CR130_LH_Rot_Cyl(
	Auto:=OP130_AutoSelected , 
	Manual:=OP130_ManualSelected, 
	ErrorActive:=OP130_ErrorActive , 
	ResetPB:= , 
	Sensor1:= I130_LH_ROTRY_180_DEGI1300_1, 
	Sensor2:= I130_LH_ROTRY_0_DEGI1300_0, 
	ManualPB1:= , 
	ManualPB2:= , 
	AutoCmd1:= , 
	AutoCmd2:= , 
	OperationEnable:=OperationEnable , 
	SafeHome:= , 
	SafeWork:= , 
	HomingCmd1:= , 
	Pulse_1Sec:=Pulse_Block.Q1Hz , 
	BlinkingBit:= , 
	TimeOut1:=10 , 
	TimeOut2:=10 , 
	TimeOut3:=10 , 
	Solenoid1=> O130_LH_ROTRY_180_DEG_Q1340_1, 
	Solenoid2=> O130_LH_ROTRY_0_DEG_Q1340_0, 
	AlarmSensor1=>berror[1201] , 
	AlarmSensor2=>berror[1202] , 
	AlarmSolenoid1=>berror[1205] , 
	AlarmSolenoid2=>berror[1206] , 
	AllSignal=>berror[1207] , 
	AlarmPresent=> , 
	Position1=> , 
	Position2=> , 
	HomeSensorBlink=> , 
	WorkSensorBlink=> , 
	Status:=CR130_LH_Rotart_Cyl_Stats );
	
//RH Rotary Cylinder


//move ZERO to STATUS
OP130_GVL.CR130_RH_Rotart_Cyl_Status:=0;



//Reset Auto Cmd IN Manual Mode & Homing
IF ( OP130_HomeRunning) THEN
	CR130_RH_Rot_Cyl.AutoCmd1:=FALSE;
	CR130_RH_Rot_Cyl.AutoCmd2:=FALSE;		
END_IF

// Safe Home
IF SR130_stManualModeAxis_RH_Vert_Servo.actualPosition >=57.0 THEN 
	CR130_RH_Rot_Cyl.SafeHome:= TRUE ;
	ELSE 
		CR130_RH_Rot_Cyl.SafeHome:= FALSE ;
	END_IF
// Safe Work
IF SR130_stManualModeAxis_RH_Vert_Servo.actualPosition >=57.0   THEN 
	CR130_RH_Rot_Cyl.Safework:= TRUE ;
	ELSE 
		CR130_RH_Rot_Cyl.Safework:= FALSE ;
	END_IF
	
// Manual PB  Cyl Mapping
IF (OP130_HMI_RH_Rotary_Cyl_Home_PB=TRUE) THEN
	CR130_RH_Rot_Cyl.ManualPB1:=TRUE;
	ELSE 
		CR130_RH_Rot_Cyl.ManualPB1:=FALSE;
	END_IF
	
IF (OP130_HMI_RH_Rotary_Cyl_Work_PB=TRUE) THEN
	CR130_RH_Rot_Cyl.ManualPB2:=TRUE;
	ELSE 
		CR130_RH_Rot_Cyl.ManualPB2:=FALSE;
	END_IF


	
CR130_RH_Rot_Cyl(
	Auto:=OP130_AutoSelected , 
	Manual:=OP130_ManualSelected , 
	ErrorActive:=OP130_ErrorActive , 
	ResetPB:= , 
	Sensor1:= I130_RH_ROTRY_180_DEGI1300_3, 
	Sensor2:= I130_RH_ROTRY_0_DEGI1300_2, 
	ManualPB1:= , 
	ManualPB2:= , 
	AutoCmd1:= , 
	AutoCmd2:= , 
	OperationEnable:=OperationEnable , 
	SafeHome:= , 
	SafeWork:= , 
	HomingCmd1:= , 
	Pulse_1Sec:=Pulse_Block.Q1Hz  , 
	BlinkingBit:= , 
	TimeOut1:=10 , 
	TimeOut2:=10 , 
	TimeOut3:=10 , 
	Solenoid1=> O130_RH_ROTRY_180_DEG_Q1340_3, 
	Solenoid2=> O130_RH_ROTRY_0_DEG_Q1340_2, 
	AlarmSensor1=>berror[1208] , 
	AlarmSensor2=>berror[1209] , 
	AlarmSolenoid1=>berror[1210] , 
	AlarmSolenoid2=>berror[1211] , 
	AllSignal=>berror[1212] , 
	AlarmPresent=> , 
	Position1=> , 
	Position2=> , 
	HomeSensorBlink=> , 
	WorkSensorBlink=> , 
	Status:=CR130_RH_Rotart_Cyl_Stats );
	
//LH Vertical Slide Servo

// Servo Safe To move
IF (SR130_stManualModeAxis_LH_Vert_Servo.actualPosition < 57.0 AND CR130_LH_Rot_Cyl.Position2)  THEN 
	OP130_LH_Servo_Safety:= FALSE;
	ELSE
	OP130_LH_Servo_Safety:= TRUE;	
	END_IF



//SR130_LH_Vert_Servo(
//	bAxis1_Ref_Switch:= , 
//	bInit:= , 
//	bErrorReset:= , 
//	bEnable:= , 
//	bMoveVelocity:= , 
//	bHalt:= , 
//	bManualMode:= , 
//	fHomePos:=SR130_LH_Servo_Control.Reference_Position , 
//	fOverride:= , 
//	fTargetPosition:= , 
//	fTargetVelocity:= , 
//	fAcc:= , 
//	fDec:= , 
//	Axis:=SR130_RH_Vert_Servo_Axis, 
//	bHome:=SR130_LH_Servo_Control.Reference_Start , 
//	bSetPosition:=SR130_LH_Servo_Control.BsetPos , 
//	bMoveAbsolute:=SR130_LH_Servo_Control.ABSmove_Start , 
//	bMoveRelative:=SR130_LH_Servo_Control.RELmove_Start , 
//	stManualModeAxis:=SR130_stManualModeAxis_LH_Vert_Servo, 
//	sAxisState=>SR130_LH_Servo_Control.Axis_State , 
//	bAxis_ready=>SR130_LH_Servo_Control.Axis_ready , 
//	bAxisInPosition=>SR130_LH_Servo_Control.Axis_In_Pos , 
//	bAxisError=>SR130_LH_Servo_Control.Axis_Error , 
//	bAxisEnabled=>SR130_LH_Servo_Control.Axis_Enabled , 
//	bAxisHomed=>SR130_LH_Servo_Control.Axis_reference , 
//	bSetPositionDone=> , 
//	bHaltDone=> , 
//	bSTOPDone=> , 
//	bHomeDone=> , 
//	bDone=> );

	
	//LH Vertical Servo 1
	SR130_LH_Vert_Servo(
	bAxis1_Ref_Switch:= , 
	bInit:= , 
	bErrorReset:=OP130_HMI_Reset OR Servo_Reset , 
	bEnable:= OperationEnable, 
	bMoveVelocity:= , 
	bHalt:= , 
	bManualMode:=OP130_ManualSelected , 
	fHomePos:= , 
	fOverride:= , 
	fTargetPosition:=SR130_LH_Servo_Control.Position , 
	fTargetVelocity:=SR130_LH_Servo_Control.Velocity, 
	fAcc:= , 
	fDec:= ,
	Servo_High_Limit:= SR130_LH_Vert_Servo_Max_Limit,	
	Servo_Low_Limit:=SR130_LH_Vert_Servo_Min_Lim,	 	
	WARNING_LIMIT:=1,
	TORQUE_LIMIT=>,	 
	Safe_move_Conditions:=OP130_LH_Servo_Safety , 
	Axis:= SR130_LH_Vert_Servo_Axis, 
	HME_WRITE_ADD:= 16#5013,	
	bHome:= SR130_LH_Servo_Control.Reference_Start, 
	bSetPosition:=SR130_LH_Servo_Control.BsetPos , 
	bMoveAbsolute:= SR130_LH_Servo_Control.ABSmove_Start , 
	bMoveRelative:=SR130_LH_Servo_Control.RELmove_Start , 
	bMoveTorque:=SR130_LH_Servo_Control.Torque_mode_Start , 
	stManualModeAxis:=SR130_stManualModeAxis_LH_Vert_Servo , 
	bmove_home:=SR130_LH_Servo_Control.Axis_Home_Cmd , 
	sAxisState=>SR130_LH_Servo_Control.Axis_State , 
	bAxis_ready=>SR130_LH_Servo_Control.Axis_ready , 
	bAxisInPosition=>SR130_LH_Servo_Control.Axis_In_Pos , 
	bAxisError=>berror[1250] , 
	bAxisEnabled=> SR130_LH_Servo_Control.Axis_Enabled, 
	bAxisHomed=>SR130_LH_Servo_Control.Axis_reference  , 
	bSetPositionDone=> , 
	bHaltDone=> SR130_LH_Servo_Control.Axis_Halted, 
	bSTOPDone=> SR130_LH_Servo_Control.Axis_Stopped, 
	bHomeDone=> , 
	bDone=> , 
	bTorqueReached=>SR130_LH_Servo_Control.Trq_reached , 
	bsafe_to_move=>SR130_LH_Servo_Control.Safe_To_Move , 
	baxis_in_home_pos=>SR130_LH_Servo_Control.Axis_In_Home , 
	bABS_Pos_done=> , 
	Actual_position=>SR130_LH_Servo_Control.Actual_Position, 
	Actual_velocity=>SR130_LH_Servo_Control.Actual_Velocity , 
	Actual_Torque=>SR130_LH_Servo_Control.Actual_Torque );
	

	
	//RH Vertical Slide Servo

// Servo Safe To move
IF (SR130_stManualModeAxis_RH_Vert_Servo.actualPosition < 57.0 AND CR130_RH_Rot_Cyl.Position2) THEN 
	OP130_RH_Servo_Safety:= FALSE;
	ELSE
	OP130_RH_Servo_Safety:= TRUE;	
	END_IF


//SR130_RH_Vert_Servo(
//	bAxis1_Ref_Switch:= , 
//	bInit:= , 
//	bErrorReset:= , 
//	bEnable:= , 
//	bMoveVelocity:= , 
//	bHalt:= , 
//	bManualMode:= , 
//	fHomePos:=SR130_RH_Servo_Control.Reference_Position , 
//	fOverride:= , 
//	fTargetPosition:= , 
//	fTargetVelocity:= , 
//	fAcc:= , 
//	fDec:= , 
//	Axis:=SR130_LH_Vert_Servo_Axis , 
//	bHome:=SR130_RH_Servo_Control.Reference_Start , 
//	bSetPosition:=SR130_RH_Servo_Control.BsetPos , 
//	bMoveAbsolute:=SR130_RH_Servo_Control.ABSmove_Start , 
//	bMoveRelative:=SR130_RH_Servo_Control.RELmove_Start , 
//	stManualModeAxis:=SR130_stManualModeAxis_RH_Vert_Servo , 
//	sAxisState=>SR130_RH_Servo_Control.Axis_State , 
//	bAxis_ready=>SR130_RH_Servo_Control.Axis_ready , 
//	bAxisInPosition=>SR130_RH_Servo_Control.Axis_In_Pos , 
//	bAxisError=>SR130_RH_Servo_Control.Axis_Error , 
//	bAxisEnabled=>SR130_RH_Servo_Control.Axis_Enabled , 
//	bAxisHomed=>SR130_RH_Servo_Control.Axis_reference , 
//	bSetPositionDone=> , 
//	bHaltDone=> , 
//	bSTOPDone=> , 
//	bHomeDone=> , 
//	bDone=> );
	
//RH Vert Servo 1

SR130_RH_Vert_Servo(
	bAxis1_Ref_Switch:= , 
	bInit:= , 
	bErrorReset:=OP130_HMI_Reset OR Servo_Reset , 
	bEnable:= OperationEnable , 
	bMoveVelocity:= , 
	bHalt:= , 
	bManualMode:=OP130_ManualSelected , 
	fHomePos:=SR130_RH_Servo_Control.Reference_Position , 
	fOverride:= , 
	fTargetPosition:= SR130_RH_Servo_Control.Position , 
	fTargetVelocity:=SR130_RH_Servo_Control.Velocity , 
	fAcc:= , 
	fDec:= ,
	Servo_High_Limit:= SR130_LH_Vert_Servo_Max_Limit,	
	Servo_Low_Limit:=SR130_LH_Vert_Servo_Min_Lim,	 	
	WARNING_LIMIT:=1,
	Actual_Torque=>SR130_RH_Servo_Control.Actual_Torque  ,
	Actual_position=> ,
    Actual_velocity=> ,
	TORQUE_LIMIT=>,	 
	Safe_move_Conditions:=OP130_RH_Servo_Safety , 
	Axis:= SR130_RH_Vert_Servo_Axis, 
	HME_WRITE_ADD:= 16#5012,	
	bHome:=SR130_LH_Servo_Control.Reference_Start , 
	bSetPosition:= SR130_RH_Servo_Control.BsetPos, 
	bMoveAbsolute:= SR130_RH_Servo_Control.ABSmove_Start, 
	bMoveRelative:=SR130_RH_Servo_Control.RELmove_Start , 
	bMoveTorque:=SR130_RH_Servo_Control.Torque_mode_Start , 
	stManualModeAxis:=SR130_stManualModeAxis_RH_Vert_Servo , 
	bmove_home:=SR130_RH_Servo_Control.Axis_Home_Cmd , 
	sAxisState=>SR130_RH_Servo_Control.Axis_State , 
	bAxis_ready=>SR130_RH_Servo_Control.Axis_ready  , 
	bAxisInPosition=>SR130_RH_Servo_Control.Axis_In_Pos , 
	bAxisError=>berror[1251] , 
	bAxisEnabled=>SR130_RH_Servo_Control.Axis_Enabled , 
	bAxisHomed=>SR130_RH_Servo_Control.Axis_reference , 
	bSetPositionDone=> , 
	bHaltDone=>SR130_RH_Servo_Control.Axis_Halted , 
	bSTOPDone=>SR130_RH_Servo_Control.Axis_Stopped , 
	bHomeDone=> , 
	bDone=> , 
	bTorqueReached=> SR130_RH_Servo_Control.Trq_reached, 
	bsafe_to_move=> SR130_RH_Servo_Control.Safe_To_Move, 
	baxis_in_home_pos=>SR130_RH_Servo_Control.Axis_In_Home , 
	bABS_Pos_done=> , 
	Actual_position=>SR130_RH_Servo_Control.Actual_Position , 
	Actual_velocity=>SR130_RH_Servo_Control.Actual_Velocity , 
	Actual_Torque=> SR130_RH_Servo_Control.Actual_Torque);
	
	// Clamping Stepper 
	// Servo Safe To move
IF (TRUE) THEN 
	SR130_RH_Servo_Control.Safe_To_Move:= TRUE;
END_IF
IF MANUAL_SELECTED THEN
	SR130_stManualModeAxis_Clamp_Stepper.targetVelocity:=50;
END_IF

SR130_Clm_Stepper(														// FESTO GUIDE GRIPPER
	bAxis1_Ref_Switch:= , 
	bInit:=  , 
	bErrorReset:=OP130_HMI_Reset OR Servo_Reset , 
	bEnable:= Servo_Enable , 
	bMoveVelocity:= , 
	bHalt:= , 
	bManualMode:=  OP130_ManualSelected, 									//MANUAL REGISTER CHANGE
	fHomePos:= , 
	fOverride:= , 
	fTargetPosition:= SR130_Stepper_Control.Position, 
	fTargetVelocity:= SR130_Stepper_Control.Velocity, 
	fAcc:= , 
	fDec:= , 
	Servo_High_Limit:= 100,	
	Servo_Low_Limit:= -100,	 	
	WARNING_LIMIT:=1,	
	Safe_move_Conditions:= Servo_Safety , 					// CHANGE
	Axis:= SR130_Clm_Stepper_Axis, 
	bHome:=SR130_Stepper_Control.Bsethome, 
	bSetPosition:= FESTO_NOT_NEED , 
	bMoveAbsolute:= SR130_Stepper_Control.ABSmove_Start, 
	bMoveRelative:= NOT_REQ , 
	bMoveTorque:= NOT_REQ , 
	stManualModeAxis:= SR130_stManualModeAxis_Clamp_Stepper, 
 	sAxisState=>SR130_Stepper_Control.Axis_State , 
	bAxis_ready=>SR130_Stepper_Control.Axis_ready , 
	bAxisInPosition=> , 
	bAxisError=> , 
	bAxisEnabled=> , 
	bAxisHomed=> , 
	bSetPositionDone=> , 
	bHaltDone=> , 
	bSTOPDone=> , 
	bHomeDone=> , 
	bDone=> , 
	bTorqueReached=> , 
	bsafe_to_move=> , 
	baxis_in_home_pos=>SR130_Stepper_Control.Axis_In_Home , 
	bABS_Pos_done=> , 
	Actual_position=>SR130_Stepper_Control.Actual_Position,
	Actual_velocity=>SR130_Stepper_Control.Actual_Velocity , 
	Actual_Torque=>SR130_Stepper_Control.Actual_Torque );

END_PROGRAM

// ---- POUs/Programs/OP130/OP130_AutoSequence.TcPOU
PROGRAM OP130_AutoSequence
VAR
	State: INT;
	OP130_Stepper_Pos : REAL:=24;
	temp5: BOOL;
	OP130_StnEnableTRIG: R_TRIG;
	dry_run:BOOL;
	fix_lh:INT;
	fix_rh:INT;
	op130_clamp_stepper_work: BOOL;
	op130_cycle_time_fb :FB_cycleTime;
	OP130_Cycle_time : UDINT;
	parts_ok: INT;
	parts_nok: INT;
END_VAR

IF (NOT OP130_Auto OR  OP130_ErrorActive OR OP130_HomeRunning OR OP130_Machine_Stop ) THEN
	OP130_GVL.OP130_AutoRunning:= FALSE;
	OP130_GVL.OP130_Home_ConditionOK:=FALSE;
	OP130_Dry_Run:=FALSE;
	OP130_ComponentOk:=FALSE;
	OP130_ComponentNok:=FALSE;
	OP130_RH_Comp_OK:=FALSE;
	OP130_RH_Comp_NOK:= FALSE;
	OP130_LH_Comp_OK:=FALSE;
	OP130_LH_Comp_NOK:= FALSE;
	OP130_AutoSeq:= 10;
	OP130_LH_AutoSeq:=0;
	OP130_RH_AutoSeq:=0;
END_IF

(*IF OP130_Auto AND NOT OP130_HomeRunning THEN
	SR130_Stepper_Control.Position:=OP130_Stepper_Pos;
	SR130_Stepper_Control.Velocity:=50;
ELSE
	SR130_Stepper_Control.Position:=0;
	SR130_Stepper_Control.Velocity:=50;
	SR130_Stepper_Control.ABSmove_Start:=1;
END_IF
*)

CASE OP130_AutoSeq OF 
	10:IF (OP130_Auto) THEN		// Check Automode Selected
		  OP130_AutoSeq :=20;
	    END_IF
		
	20:IF ( NOT OP130_ErrorActive) THEN		//Check No error
		  OP130_AutoSeq:=30;
	   END_IF
	   
	30:IF (NOT OP130_HomeRunning) THEN		//Check No Homerunning
		  OP130_AutoSeq :=40;
		END_IF
		
    40:IF ( OP130_GVL.OP130_Temp_Home_OK)THEN	//Check Machine in Home
		  OP130_AutoSeq:= 50;
		END_IF
		
	50:IF ( NOT OP130_OperationCompleted) THEN		// Check Operation Completed Reset
		OP130_AutoSeq:=60;
		END_IF
		
	60:IF (NOT OP130_ComponentOk) THEN		// Check Component Ok Reset
		OP130_AutoSeq:=70;
		END_IF
		
	70:IF (NOT OP130_ComponentNok) THEN 	// Check Component NOk Reset
		OP130_AutoSeq:= 120;
		END_IF
		
    120:IF  (OP130_HMI_Cycle_Start OR OP130_Dry_Run) THEN		//Machine Start in Fully Automatic or Press Cycle Start For Semi Automatic
		    OP130_GVL.OP130_Home_ConditionOK:=TRUE;
	 			IF( OP130_GVL.OP130_Home_ConditionOK AND OP130_AutoSelected) THEN
					OP130_AutoRunning:=TRUE;
					OP130_StepRunning:= FALSE;
				
				ELSIF (OP130_Home_ConditionOK AND OP130_StepSelected) THEN
					OP130_AutoRunning:=FALSE;
					OP130_StepRunning:= TRUE;
				END_IF;
		 END_IF
		 IF ((OP130_AutoRunning OR OP130_StepRunning) AND OP130_StartEnable) THEN
			     SR130_Stepper_Control.ABSmove_Start:=1;
				 OP130_AutoSeq:= 130;
		END_IF
	130:IF (OP130_StartEnable) THEN // Check Previous Station Completed
				OP130_AutoSeq:= 131;       
     	END_IF
	
     131:   SR130_Stepper_Control.Position:=88;
            SR130_Stepper_Control.Velocity:=50;
		    SR130_Stepper_Control.ABSmove_Start:=TRUE;
             IF SR130_Clm_Stepper.bAxisInPosition AND op130_clamp_stepper_work THEN
				SR130_Stepper_Control.ABSmove_Start:=FALSE; 
		        OP130_AutoSeq:= 140;
		     END_IF
	 	
	140: IF NOT OP130_STN_ENABLE AND MOVER_POS_RECHED[OP130_STN_MOVER] AND fix_lh <> 120 AND fix_rh <> 120 THEN
         	OP130_AutoSeq:= 200;
         ELSIF OP130_STN_ENABLE AND fix_lh =120 AND fix_rh =120 THEN
           OP130_Prev_LH_COMP_OK:=TRUE;
	       OP130_Prev_RH_COMP_OK:=TRUE;
           OP130_Prev_LH_COMP_NOK:=FALSE;
           OP130_Prev_RH_COMP_NOK:=FALSE;
		   OP130_AutoSeq:= 141;
         ELSIF OP130_STN_ENABLE AND fix_lh = 120 AND fix_rh =121 THEN
           OP130_Prev_LH_COMP_OK:=TRUE;
	       OP130_Prev_RH_COMP_OK:=FALSE;
           OP130_Prev_LH_COMP_NOK:=FALSE;
           OP130_Prev_RH_COMP_NOK:=TRUE;
		   OP130_AutoSeq:= 141;
         ELSIF OP130_STN_ENABLE AND fix_lh = 121 AND fix_rh =120 THEN
           OP130_Prev_LH_COMP_OK:=false;
	       OP130_Prev_RH_COMP_OK:=TRUE;
		   OP130_Prev_LH_COMP_NOK:=TRUE;
           OP130_Prev_RH_COMP_NOK:=FALSE;
           OP130_AutoSeq:= 141;
          END_IF 
		  
    141:	OP130_LH_AutoSeq:=10;
            OP130_RH_AutoSeq:=10;
		    OP130_AutoSeq:= 150;  
		  
   
	150:IF (OP130_LH_Operation_Completed AND OP130_RH_Operation_Completed ) THEN	//Waiting For Both RH & LH Seq Completion
			OP130_MVR_DN_PERMISSION			:= TRUE;
			OP130_AutoSeq					:= 151;			
		 END_IF
		 OP130_CURR_MOVER		:=OP130_STN_MOVER;
	
	151: IF NOT OP130_MVR_DN_PERMISSION THEN
			OP130_AutoSeq					:= 155;		
		END_IF	 
	
	155:IF OP130_LH_Comp_OK AND OP130_rH_Comp_OK THEN
				MOVER_CMP_STATUS[OP130_CURR_MOVER][1]:=130;	
                MOVER_CMP_STATUS[OP130_CURR_MOVER][2]:=130;
		            IF MOVER_CMP_STATUS[OP130_CURR_MOVER][1]=130 AND MOVER_CMP_STATUS[OP130_CURR_MOVER][2]=130 THEN
			     	STATION_DONE[OP130_CURR_MOVER][OP130_XTS_POS_NO]			:= TRUE;
			            OP130_AutoSeq:= 160;
						parts_ok :=parts_ok+1;
				     END_IF
				ELSIF OP130_LH_Comp_NOK AND OP130_rH_Comp_OK THEN	
					  MOVER_CMP_STATUS[OP130_CURR_MOVER][1]:=130;	
                      MOVER_CMP_STATUS[OP130_CURR_MOVER][2]:=130;
		               IF MOVER_CMP_STATUS[OP130_CURR_MOVER][1]=130 AND MOVER_CMP_STATUS[OP130_CURR_MOVER][2]=130 THEN
			         	STATION_DONE[OP130_CURR_MOVER][OP130_XTS_POS_NO]			:= TRUE;
			              OP130_AutoSeq:= 160;
						  parts_nok :=parts_nok+1;
			    	   END_IF
                 ELSIF OP130_LH_Comp_OK AND OP130_rH_Comp_NOK THEN	
					  MOVER_CMP_STATUS[OP130_CURR_MOVER][1]:=130;	
                      MOVER_CMP_STATUS[OP130_CURR_MOVER][2]:=130;
		               IF MOVER_CMP_STATUS[OP130_CURR_MOVER][1]=130 AND MOVER_CMP_STATUS[OP130_CURR_MOVER][2]=130 THEN
			       	STATION_DONE[OP130_CURR_MOVER][OP130_XTS_POS_NO]			:= TRUE;
			              OP130_AutoSeq:= 160;
						  parts_nok :=parts_nok+1;
			    	   END_IF	
					   ELSIF OP130_LH_Comp_NOK AND OP130_rH_Comp_NOK THEN	
					  MOVER_CMP_STATUS[OP130_CURR_MOVER][1]         :=130;	
                      MOVER_CMP_STATUS[OP130_CURR_MOVER][2]         :=130;
		               IF MOVER_CMP_STATUS[OP130_CURR_MOVER][1]=130 AND MOVER_CMP_STATUS[OP130_CURR_MOVER][2]=130 THEN
			          	STATION_DONE[OP130_CURR_MOVER][OP130_XTS_POS_NO]			:= TRUE;
			              OP130_AutoSeq:= 160;
						  parts_nok :=parts_nok+1;
					   END_IF
			  END_IF	
		
	160:IF ( OP130_StartEnable) THEN  // Operation Completed
	        OP130_Cycle_Time_Stop                                   :=TRUE;
			OP130_OperationCompleted                                :=TRUE;
			OP130_AutoSeq                                           := 170;
			STATION_DONE[OP130_CURR_MOVER][OP130_XTS_POS_NO]			:= TRUE;
		END_IF
		
	170:OP130_LH_Operation_Completed             :=FALSE;
	    OP130_RH_Operation_Completed             :=FALSE;
	    OP130_OperationCompleted                 :=FALSE;
	    OP130_ComponentOk                        :=FALSE;
	    OP130_ComponentNOk                       :=FALSE;
	    OP130_AutoSeq                            :=180;
	
	(*171 : SR130_Stepper_Control.Position:=0;
          SR130_Stepper_Control.Velocity:=50;
		  SR130_Stepper_Control.ABSmove_Start:=TRUE;
		  
             IF SR130_Clm_Stepper.bAxisInPosition THEN
				SR130_Stepper_Control.ABSmove_Start:=FALSE; 
		        OP130_AutoSeq:= 180;
		     END_IF*)
	
	180:		// Reset All Bits	
	
        OP130_Prev_LH_COMP_OK:=FALSE;
		OP130_Prev_RH_COMP_OK:=FALSE;						
        OP130_LH_Comp_OK:=FALSE;
        OP130_LH_Comp_NOK:=FALSE;
        OP130_RH_Comp_OK:=FALSE;
        OP130_RH_Comp_NOK:=FALSE;
        OP130_LH_AutoSeq:=0;
		OP130_RH_AutoSeq:=0;
		OP130_AutoSeq:= 130;
		
		
   200:	MOVER_CMP_STATUS[OP130_CURR_MOVER][1]:=130;	 ///// NEED TO BE UPDATED AS 131
        MOVER_CMP_STATUS[OP130_CURR_MOVER][2]:=130;
		IF MOVER_CMP_STATUS[OP130_CURR_MOVER][1]=130 AND MOVER_CMP_STATUS[OP130_CURR_MOVER][2]=130 THEN
				STATION_DONE[OP130_CURR_MOVER][OP130_XTS_POS_NO]			:= TRUE;
			OP130_AutoSeq:= 180;
		END_IF


END_CASE

op130_cycle_time_fb(i_b_startTime:=OP130_STN_ENABLE , i_b_stopTime:= NOT OP130_STN_ENABLE , o_t_StationTime=>OP130_Cycle_time );
dry_run:=All_Station_Dry_Run;
//staus FOR movers 
IF  dry_run THEN
	fix_lh :=120;
	fix_rh :=120;
ELSE 
	fix_lh := MOVER_CMP_STATUS[OP130_STN_MOVER][1];
	fix_rh := MOVER_CMP_STATUS[OP130_STN_MOVER][2];
END_IF

op130_clamp_stepper_work:=In_Range(value:=SR130_Clm_Stepper.Actual_position, setvalue:= 88, tolerance:= 0.2);



//############################		OP130 STATION ENABLE CONDITION		##########################

	OP130_STN_MOVER					:= MOVER_POSITION[OP130_XTS_POS_NO];
	IF AUTO_WITH_XTS THEN
	IF OP130_STN_MOVER>0 THEN
	IF NOT(END_OF_CYCLE AND MOVER_CMP_STATUS[OP130_STN_MOVER][1]=5 AND MOVER_CMP_STATUS[OP130_STN_MOVER][2]=5)THEN		
	OP130_STN_ENABLE				:= MOVER_POS_RECHED[OP130_STN_MOVER] AND ((MOVER_CMP_STATUS[OP130_STN_MOVER][1]=120)OR 
										(MOVER_CMP_STATUS[OP130_STN_MOVER][2]=120))AND STATION_ENABLE_CONTROL;		
	ELSE
	STATION_DONE[OP130_STN_MOVER][OP130_XTS_POS_NO]			:= TRUE;		
	END_IF
	ELSE
	OP130_STN_ENABLE				:= FALSE;	
	END_IF
	END_IF

END_PROGRAM

// ---- POUs/Programs/OP130/OP130_LH_Auto.TcPOU
PROGRAM OP130_LH_Auto
VAR
	OP130_Torque_Monitor_Dly: TON;
	Temp1:BOOL;
	act_torque:LREAL;
END_VAR

CASE OP130_LH_AutoSeq OF
	10: IF (OP130_Prev_LH_COMP_OK= TRUE) AND OP130_StartEnable THEN   //Check LH Comp OK
		OP130_LH_AutoSeq:=20;
		END_IF
		IF (OP130_Prev_LH_COMP_NOK= TRUE) THEN 
			OP130_LH_AutoSeq:=180;
		END_IF
	
	20:IF  OP130_StartEnable THEN	// Check Mover Presence in Station
		   OP130_LH_AutoSeq:=30;
	   END_IF
	   
	30:IF (OP130_GVL.SR130_LH_Servo_Control.Axis_Enabled=TRUE OR OP130_Dry_Run) AND OP130_StartEnable THEN // Check Servo Axis Enabled
		   OP130_LH_AutoSeq:=40;
		END_IF
		
	40:IF  OP130_StartEnable THEN  // Check Rotary Cyl In Zero Deg
		   OP130_LH_AutoSeq:=50;
	   END_IF
	   
	50:IF OP130_StartEnable THEN 		//Move Work Position Value to Servo
		//  OP130_GVL.SR130_LH_Vert_Servo.fTargetPosition:=SR130_HMI_Servo_Work_Position;
		//  OP130_GVL.SR130_LH_Vert_Servo.fTargetVelocity:=SR130_HMI_Servo_Work_Velocity;
		SR130_LH_Servo_Control.Position:=SR130_HMI_Servo_Work_Position;
		SR130_LH_Servo_Control.Velocity:=SR130_HMI_Servo_Work_Velocity;
		OP130_LH_AutoSeq:=60;
		END_IF
		
	60:IF OP130_StartEnable THEN 	//Move Cmd to Servo
		//SR130_LH_Abs_Move_Start:=TRUE;
		SR130_LH_Servo_Control.ABSmove_Start:=TRUE;
		OP130_LH_AutoSeq:=70;
		END_IF
		
	70:IF OP130_StartEnable AND OP130_GVL.SR130_LH_Servo_Control.Axis_In_Pos THEN // Check Servo in Target Pos
		//SR130_LH_Abs_Move_Start:=FALSE;
		SR130_LH_Servo_Control.ABSmove_Start:=FALSE;
		OP130_LH_AutoSeq:=90;
		END_IF
	
	90:IF OP130_StartEnable THEN		//Move Lock Position Value to Servo
		//OP130_GVL.SR130_LH_Vert_Servo.fTargetPosition:=SR130_HMI_Servo_Lock_Position;
		//OP130_GVL.SR130_LH_Vert_Servo.fTargetVelocity:=SR130_HMI_Servo_Lock_Velocity;
	     SR130_LH_Servo_Control.Position:=SR130_HMI_Servo_Lock_Position;
		 SR130_LH_Servo_Control.Velocity:=SR130_HMI_Servo_Lock_Velocity;
		 OP130_LH_AutoSeq:=100;
		 END_IF
		 
	100:IF OP130_StartEnable THEN		// MOve Cmd to Servo
		//SR130_LH_Abs_Move_Start:=TRUE;
		   SR130_LH_Servo_Control.ABSmove_Start :=TRUE;
		   OP130_LH_AutoSeq:=110;
		END_IF
		
    110:IF OP130_StartEnable  THEN		//Check Servo In Target Pos
		IF SR130_LH_Servo_Control.Axis_In_Pos AND SR130_LH_Servo_Control.Actual_Torque < OP130_HMI_Pull_Torque_Limit THEN
			act_torque:=SR130_LH_Servo_Control.Actual_Torque;
			SR130_LH_Vert_Servo.bHalt:=TRUE;
			OP130_LH_Comp_OK:=TRUE;
			OP130_LH_Comp_NOK:= FALSE;
	//	SR130_LH_Abs_Move_Start:=FALSE;
		SR130_LH_Servo_Control.ABSmove_Start:=FALSE;
		END_IF
		IF SR130_LH_Servo_Control.Axis_In_Pos AND SR130_LH_Servo_Control.Actual_Torque > OP130_HMI_Pull_Torque_Limit THEN
			OP130_LH_Comp_NOK:=TRUE;
			OP130_LH_Comp_OK:= FALSE;
			//SR130_LH_Abs_Move_Start:=FALSE;
			SR130_LH_Servo_Control.ABSmove_Start:=FALSE;
		END_IF
	    IF SR130_LH_Servo_Control.Axis_Halted OR SR130_LH_Servo_Control.Axis_In_Pos AND (OP130_LH_Comp_OK OR OP130_LH_Comp_NOK) THEN
	    //SR130_LH_Abs_Move_Start:=FALSE;
		SR130_LH_Servo_Control.ABSmove_Start:=FALSE;
        OP130_LH_AutoSeq:=180;
	    END_IF
        END_IF
	
		

	
	180:IF (OP130_StartEnable) THEN   // Move Work Pos Values to Servo
		//OP130_GVL.SR130_LH_Vert_Servo.fTargetPosition:=SR130_HMI_Servo_CylWork_Position;
       // OP130_GVL.SR130_LH_Vert_Servo.fTargetVelocity:=SR130_HMI_Servo_CylWork_Velocity;
		SR130_LH_Servo_Control.position:=SR130_HMI_Servo_CylWork_Position;
		SR130_LH_Servo_Control.velocity:=SR130_HMI_Servo_CylWork_Velocity;
		SR130_LH_Vert_Servo.bHalt:=FALSE;
        MOVER_CMP_STATUS[OP130_STN_MOVER][1]:=130;
        OP130_LH_AutoSeq:=190;
	   END_IF
	   
	 190: IF(OP130_StartEnable) THEN		//move Cmd to Servo
		// SR130_LH_Abs_Move_Start:= TRUE;
		 SR130_LH_Servo_Control.ABSmove_Start := TRUE;
		 OP130_LH_AutoSeq:=200;
	 END_IF
	 
	200:IF (OP130_StartEnable) AND OP130_GVL.SR130_LH_Servo_Control.Axis_In_Pos THEN		//Check Servo In Target Pos
	       //SR130_LH_Abs_Move_Start:= FALSE;	
		   SR130_LH_Servo_Control.ABSmove_Start := FALSE;
           OP130_LH_AutoSeq:=210;
	    END_IF
		
	210:IF  (OP130_StartEnable) THEN		//Move Rotary Cyl to Zero Deg
		    OP130_GVL.CR130_LH_Rot_Cyl.AutoCmd2:=TRUE;
		    OP130_GVL.CR130_LH_Rot_Cyl.AutoCmd1:=FALSE;
		    IF (OP130_GVL.CR130_LH_Rot_Cyl.Position2=TRUE) THEN
			   OP130_LH_AutoSeq:=220;
			   END_IF
	    END_IF
		
	220: IF  (OP130_StartEnable) THEN		//move Home Pos to Servo
		    // OP130_GVL.SR130_LH_Vert_Servo.fTargetPosition:=SR130_HMI_Servo_Rotation_Position;
		    // OP130_GVL.SR130_LH_Vert_Servo.fTargetVelocity:=SR130_HMI_Servo_Rotation_Velocity;
			 SR130_LH_Servo_Control.Position :=SR130_HMI_Servo_Rotation_Position;
			 SR130_LH_Servo_Control.Velocity :=SR130_HMI_Servo_Rotation_Velocity;
		     OP130_LH_AutoSeq:=230;
	      END_IF
	
	230: IF (OP130_StartEnable) THEN 		//Move Cmd TO Servo
		   // SR130_LH_Abs_Move_Start:= TRUE ;
			SR130_LH_Servo_Control.ABSmove_Start:= TRUE;
		    OP130_LH_AutoSeq:=240;
	     END_IF
	
	240: IF (OP130_StartEnable) AND OP130_GVL.SR130_LH_Servo_Control.Axis_In_Pos THEN 	//Check Servo In Target Pos
		    //SR130_LH_Abs_Move_Start:= FALSE ;
			SR130_LH_Servo_Control.ABSmove_Start:= FALSE;
			OP130_LH_AutoSeq:=250;
	     END_IF
	
	250:IF  (OP130_StartEnable) THEN		//Move Rotary Cyl to Zero Deg
		    OP130_GVL.CR130_LH_Rot_Cyl.AutoCmd1:=TRUE;
		    OP130_GVL.CR130_LH_Rot_Cyl.AutoCmd2:=FALSE;
		   IF (OP130_GVL.CR130_LH_Rot_Cyl.Position1=TRUE) THEN
			  OP130_LH_AutoSeq:=260;
		   END_IF
	    END_IF
		
	260: IF  (OP130_StartEnable) THEN		//move Home Pos to Servo
		     //OP130_GVL.SR130_LH_Vert_Servo.fTargetPosition:=SR130_Servo_Home_Position;
		    // OP130_GVL.SR130_LH_Vert_Servo.fTargetVelocity:=SR130_Servo_Home_Velocity;
			 SR130_LH_Servo_Control.Position := SR130_Servo_Home_Position;
			 SR130_LH_Servo_Control.Velocity := SR130_Servo_Home_Velocity;
		     OP130_LH_AutoSeq:=270;
	     END_IF
		 
	270: IF (OP130_StartEnable) THEN 		//Move Cmd TO Servo
		   // SR130_LH_Abs_Move_Start:= TRUE ;
			SR130_LH_Servo_Control.ABSmove_Start := TRUE;
		    OP130_LH_AutoSeq:=280;
	     END_IF
	
	280: IF (OP130_StartEnable) AND OP130_GVL.SR130_LH_Servo_Control.Axis_In_Pos THEN 	//Check Servo In Target Pos
		   // SR130_LH_Abs_Move_Start:= FALSE ;
			SR130_LH_Servo_Control.ABSmove_Start := FALSE;
			OP130_LH_AutoSeq:=290;
	     END_IF
		 
	 290:IF (OP130_StartEnable) THEN		//LH Operation completed
		    OP130_LH_Operation_Completed:= TRUE;
		    OP130_LH_AutoSeq:=300;
	     END_IF

	   
END_CASE
//Torque Monitor Delay
OP130_Torque_Monitor_Dly(IN:=OP130_LH_AutoSeq=170 , PT:=T#200MS , Q=> , ET=> );

END_PROGRAM

// ---- POUs/Programs/OP130/OP130_RH_Auto.TcPOU
PROGRAM OP130_RH_Auto
VAR
	OP130_Torque_Monitor_Dly: TON;
	OP130_Torque_Monitor_Dly_RH: TON;
	Temp2:BOOL;
	actual_torque:LREAL;
END_VAR

CASE OP130_RH_AutoSeq OF
	10: IF (OP130_Prev_RH_COMP_OK= TRUE) AND OP130_StartEnable THEN 
		OP130_RH_AutoSeq:=20;
		END_IF
		IF (OP130_Prev_RH_COMP_NOK= TRUE) THEN 
			OP130_RH_AutoSeq:=180;
		END_IF
	
	20:IF  OP130_StartEnable THEN	
		OP130_RH_AutoSeq:=30;
	   END_IF
	   
	30:IF (OP130_GVL.SR130_RH_Servo_Control.Axis_Enabled=TRUE OR OP130_Dry_Run) AND OP130_StartEnable THEN
		OP130_RH_AutoSeq:=40;
		END_IF
		
	40:IF  OP130_StartEnable THEN
		OP130_RH_AutoSeq:=50;
		END_IF
		
	50:IF (OP130_StartEnable) THEN 
		//OP130_GVL.SR130_RH_Vert_Servo.fTargetPosition:=SR130_HMI_Servo_Work_Position;
		//OP130_GVL.SR130_RH_Vert_Servo.fTargetVelocity:=SR130_HMI_Servo_Work_Velocity;
		SR130_RH_Servo_Control.Position :=SR130_HMI_Servo_Work_Position;
		SR130_RH_Servo_Control.Velocity :=SR130_HMI_Servo_Work_Velocity;
		OP130_RH_AutoSeq:=60;
		END_IF
		
	60:IF(OP130_StartEnable) THEN 
		//SR130_RH_Abs_Move_Start:=TRUE;
		SR130_RH_Servo_Control.ABSmove_Start:=TRUE;
		OP130_RH_AutoSeq:=70;
		END_IF
		
	70:IF(OP130_StartEnable)AND OP130_GVL.SR130_RH_Servo_Control.Axis_In_Pos THEN 
		//SR130_RH_Abs_Move_Start:=FALSE;
		SR130_RH_Servo_Control.ABSmove_Start:=FALSE;
		OP130_RH_AutoSeq:=90;
		END_IF
	
	90:IF (OP130_StartEnable) THEN
		//OP130_GVL.SR130_RH_Vert_Servo.fTargetPosition:=SR130_HMI_Servo_Lock_Position;
		//OP130_GVL.SR130_RH_Vert_Servo.fTargetVelocity:=SR130_HMI_Servo_Lock_Velocity;
		 SR130_RH_Servo_Control.Position :=SR130_HMI_Servo_Lock_Position;
		 SR130_RH_Servo_Control.Velocity :=SR130_HMI_Servo_Lock_Velocity;
		 OP130_RH_AutoSeq:=100;
		 END_IF
		 
	100:IF (OP130_StartEnable) THEN
		//SR130_RH_Abs_Move_Start:=TRUE;
		SR130_RH_Servo_Control.ABSmove_Start:=TRUE;
		 OP130_RH_AutoSeq:=110;
		END_IF
		
    110:IF OP130_StartEnable  THEN		//Check Servo In Target Pos
		IF SR130_RH_Servo_Control.Axis_In_Pos AND SR130_RH_Servo_Control.Actual_Torque < OP130_HMI_Pull_Torque_Limit THEN
			actual_torque :=SR130_RH_Servo_Control.Actual_Torque;
			SR130_RH_Vert_Servo.bHalt:=TRUE;
			OP130_RH_Comp_OK:=TRUE;
			OP130_RH_Comp_NOK:= FALSE;
		//SR130_RH_Abs_Move_Start:=FALSE;
		SR130_RH_Servo_Control.ABSmove_Start:=FALSE;
		END_IF
		IF SR130_RH_Servo_Control.Axis_In_Pos AND SR130_RH_Servo_Control.Actual_Torque > OP130_HMI_Pull_Torque_Limit THEN
			OP130_RH_Comp_NOK:=TRUE;
			OP130_RH_Comp_OK:= FALSE;
			//SR130_RH_Abs_Move_Start:=FALSE;
			SR130_RH_Servo_Control.ABSmove_Start:=FALSE;
		END_IF
	 IF SR130_RH_Servo_Control.Axis_Halted OR SR130_RH_Servo_Control.Axis_In_Pos AND (OP130_RH_Comp_OK OR OP130_RH_Comp_NOK) THEN
	//SR130_RH_Abs_Move_Start:=FALSE;
	    SR130_RH_Servo_Control.ABSmove_Start:=FALSE;
        OP130_RH_AutoSeq:=180;
		END_IF
		END_IF
	
		

	
	180:IF (OP130_StartEnable) THEN   // Move Work Pos Values to Servo
		//OP130_GVL.SR130_RH_Vert_Servo.fTargetPosition:=SR130_HMI_Servo_CylWork_Position;
		//OP130_GVL.SR130_RH_Vert_Servo.fTargetVelocity:=SR130_HMI_Servo_CylWork_Velocity;
		    SR130_RH_Servo_Control.Position :=SR130_HMI_Servo_CylWork_Position;
		    SR130_RH_Servo_Control.Velocity :=SR130_HMI_Servo_CylWork_Velocity;
		    SR130_RH_Vert_Servo.bHalt:=FALSE;
		    MOVER_CMP_STATUS[OP130_STN_MOVER][2]:=130;
            OP130_RH_AutoSeq:=190;
	   END_IF
	   
	 190: IF(OP130_StartEnable) THEN		//move Cmd to Servo
		// SR130_RH_Abs_Move_Start:= TRUE;
		 SR130_RH_Servo_Control.ABSmove_Start:= TRUE;
		 OP130_RH_AutoSeq:=200;
	 END_IF
	 
	200:IF (OP130_StartEnable) AND OP130_GVL.SR130_RH_Servo_Control.Axis_In_Pos THEN		//Check Servo In Target Pos
	       //SR130_RH_Abs_Move_Start:= FALSE;	
	       SR130_RH_Servo_Control.ABSmove_Start:= FALSE;
           OP130_RH_AutoSeq:=210;
	    END_IF
		
	210:IF  (OP130_StartEnable) THEN		//Move Rotary Cyl to Zero Deg
		OP130_GVL.CR130_RH_Rot_Cyl.AutoCmd2:=TRUE;
		  OP130_GVL.CR130_RH_Rot_Cyl.AutoCmd1:=FALSE;
		  IF (OP130_GVL.CR130_RH_Rot_Cyl.Position2=TRUE) THEN
			  OP130_RH_AutoSeq:=220;
			  END_IF
	END_IF
	
	220: IF  (OP130_StartEnable) THEN		//move Home Pos to Servo
		//OP130_GVL.SR130_RH_Vert_Servo.fTargetPosition:=SR130_HMI_Servo_Rotation_Position;
		//OP130_GVL.SR130_RH_Vert_Servo.fTargetVelocity:=SR130_HMI_Servo_Rotation_Velocity;
		      SR130_RH_Servo_Control.Position:=SR130_HMI_Servo_Rotation_Position;
		      SR130_RH_Servo_Control.Velocity:=SR130_HMI_Servo_Rotation_Velocity;
		      OP130_RH_AutoSeq:=230;
	     END_IF
	
	230: IF (OP130_StartEnable) THEN 		//Move Cmd TO Servo
		//SR130_RH_Abs_Move_Start:= TRUE ;
		SR130_RH_Servo_Control.ABSmove_Start:= TRUE ;
		 OP130_RH_AutoSeq:=240;
	     END_IF
	
	240: IF (OP130_StartEnable) AND OP130_GVL.SR130_RH_Servo_Control.Axis_In_Pos THEN 	//Check Servo In Target Pos
		// SR130_RH_Abs_Move_Start:= FALSE ;
		 SR130_RH_Servo_Control.ABSmove_Start:= FALSE ;
			OP130_RH_AutoSeq:=250;
	      END_IF
		  
	250:IF (OP130_StartEnable) THEN		//Move Rotary Cyl to Zero Deg
		   OP130_GVL.CR130_RH_Rot_Cyl.AutoCmd1:=TRUE;
		  OP130_GVL.CR130_RH_Rot_Cyl.AutoCmd2:=FALSE;
		  IF (OP130_GVL.CR130_RH_Rot_Cyl.Position1=TRUE) THEN
			  OP130_RH_AutoSeq:=260;
		  END_IF
	    END_IF
		
	260: IF  (OP130_StartEnable) THEN		//move Home Pos to Servo
		//OP130_GVL.SR130_RH_Vert_Servo.fTargetPosition:=SR130_Servo_Home_Position;
		//OP130_GVL.SR130_RH_Vert_Servo.fTargetVelocity:=SR130_Servo_Home_Velocity;
		     SR130_RH_Servo_Control.Position:=SR130_Servo_Home_Position;
		     SR130_RH_Servo_Control.Velocity:=SR130_Servo_Home_Velocity;
		     OP130_RH_AutoSeq:=270;
	     END_IF
		 
	270: IF (OP130_StartEnable) THEN 		//Move Cmd TO Servo
		//SR130_RH_Abs_Move_Start:= TRUE ;
		SR130_RH_Servo_Control.ABSmove_Start:= TRUE ;
		 OP130_RH_AutoSeq:=280;
	     END_IF
	
	280: IF (OP130_StartEnable) AND OP130_GVL.SR130_RH_Servo_Control.Axis_In_Pos THEN 	//Check Servo In Target Pos
		// SR130_RH_Abs_Move_Start:= FALSE ;
		 SR130_RH_Servo_Control.ABSmove_Start:= FALSE ;
			OP130_RH_AutoSeq:=290;
	     END_IF
		 
	 290:IF (OP130_StartEnable) THEN		//LH Operation completed
		    OP130_RH_Operation_Completed:= TRUE;
		    OP130_RH_AutoSeq:=300;
	     END_IF

	   
END_CASE
//Torque Monitor Dly
 OP130_Torque_Monitor_Dly_RH(IN:=OP130_RH_AutoSeq=170 , PT:=T#200MS , Q=> , ET=> );

END_PROGRAM

// ---- POUs/Programs/OP130/OP130_Error.TcPOU
PROGRAM OP130_Error
VAR
	OP130_StErr_1: TON;
	OP130_Step_Err_2: TON;
	end: INT;
	OP130_StepErr_3: TON;
	OP130_StErr_4: TON;
	OP130_Step_Err_5: TON;
	OP130_StepErr_6: TON;
	bdone: BOOL;
	i: INT;
	j: INT;
END_VAR


IF NOT bdone THEN
	bdone:=TRUE;
FOR i:=1200 TO 1300 BY 1 DO 
	
IF berror[i] THEN
	OP130_ErrorActive:=TRUE;
END_IF
END_FOR
bdone:=FALSE;
END_IF

IF OP130_HMI_Reset OR Servo_Reset THEN
	FOR j:=1200 TO 1300 BY 1 DO 
		
	
	berror[j]:=FALSE;
	OP130_ErrorActive:=FALSE;
	
	END_FOR
	temp:=false;
END_IF

END_PROGRAM

// ---- POUs/Programs/OP130/OP130_Initialization_Seq.TcPOU
PROGRAM OP130_Initialization_Seq
VAR
	temp3: BOOL;
END_VAR

IF OP130_LH_HomeOK AND OP130_GVL.SR130_Stepper_Control.Axis_In_Home AND OP130_RH_HomeOK THEN
   OP130_Temp_Home_OK:=TRUE;
   OP130_HomeRunning:=FALSE;
ELSE
	OP130_Temp_Home_OK:=FALSE;	
END_IF

IF (OP130_GVL.SR130_LH_Servo_Control.Axis_In_Home AND OP130_GVL.CR130_LH_Rot_Cyl.Position1 AND SR130_Clm_Stepper.bHomeDone AND SR130_Clm_Stepper.baxis_in_home_pos) THEN
	OP130_LH_HomeOK:=TRUE;
	OP130_Homing_Seq:=0;
ELSE
	OP130_LH_HomeOK:=FALSE;
END_IF

IF (OP130_GVL.SR130_RH_Servo_Control.Axis_In_Home AND OP130_GVL.CR130_RH_Rot_Cyl.Position1) THEN
	OP130_RH_HomeOK:=TRUE;
	OP130_RH_Homing_Seq:=0;
ELSE
	OP130_RH_HomeOK:=FALSE;
END_IF
	
CASE OP130_Homing_Seq OF
	
	0: IF (OP130_Auto AND NOT OP130_HomeRunning AND  NOT OP130_ErrorActive AND  NOT OP130_AutoRunning AND NOT OP130_StepRunning AND NOT OP130_Temp_Home_OK	) THEN
		OP130_HomeRunning:=TRUE;
		OP130_Homing_Seq:=10;
        OP130_RH_Homing_Seq:=10;	
	   END_IF
	   
	   10:IF SR130_stManualModeAxis_LH_Vert_Servo.actualPosition >=61  THEN
		  OP130_Homing_Seq:=20;
	      ELSE
		   OP130_Homing_Seq:=90;
		  END_IF
	   
	   20: IF (OP130_HomeRunning AND OP130_HMI_Homing)THEN 
		    
			  SR130_LH_Servo_Control.Position :=SR130_HMI_Servo_CylWork_Position;
			  SR130_LH_Servo_Control.velocity :=SR130_HMI_Servo_CylWork_Velocity;
		      OP130_Homing_Seq:=30;
	   END_IF
	   
	   30: IF (OP130_HomeRunning AND OP130_HMI_Homing)THEN 
		    
			SR130_LH_Servo_Control.ABSmove_Start := TRUE;
			 OP130_Homing_Seq:=35;
	   END_IF
	   
	   35 : IF (OP130_HomeRunning AND OP130_HMI_Homing)THEN 
		   	   SR130_Stepper_Control.Bsethome:=1;
			   IF SR130_Stepper_Control.Axis_In_Home THEN
				  OP130_Homing_Seq:=40; 
			   END_IF
	        END_IF
	   
	   40:IF (OP130_HomeRunning AND OP130_HMI_Homing)THEN 
		   IF OP130_GVL.SR130_LH_Servo_Control.Axis_In_Pos THEN
			 SR130_LH_Servo_Control.ABSmove_Start := FALSE;
			 OP130_Homing_Seq:=50;
		   END_IF
	      END_IF
	   
	   50:IF (OP130_HomeRunning AND OP130_HMI_Homing)THEN 
		   IF CR130_LH_Rot_Cyl.Position2 THEN
			   OP130_Homing_Seq:=60; 
		  ELSE
		   OP130_GVL.CR130_LH_Rot_Cyl.HomingCmd2:= TRUE;
		   OP130_GVL.CR130_LH_Rot_Cyl.HomingCmd1:= FALSE;
	      END_IF
	      END_IF
		  
	   60:IF (OP130_HomeRunning AND OP130_HMI_Homing)THEN 
		    
			 SR130_LH_Servo_Control.Position := SR130_HMI_Servo_Rotation_Position;
			 SR130_LH_Servo_Control.Velocity := SR130_HMI_Servo_Rotation_Velocity;
		     OP130_Homing_Seq:=70;
	      END_IF
		  
	   70: IF (OP130_HomeRunning AND OP130_HMI_Homing)THEN 
		     
		      SR130_LH_Servo_Control.ABSmove_Start := TRUE;
			  OP130_Homing_Seq:=75;
			 END_IF
	   
	   75:IF  OP130_GVL.SR130_LH_Servo_Control.Axis_In_Pos THEN 
		      SR130_LH_Servo_Control.ABSmove_Start := FALSE;
              OP130_Homing_Seq:=80;
	      END_IF
	   
	   
	   80:IF (OP130_HomeRunning AND OP130_HMI_Homing)THEN 
		      IF OP130_GVL.CR130_LH_Rot_Cyl.Position1 THEN
			     OP130_Homing_Seq:=90;
			   ELSE
				OP130_GVL.CR130_LH_Rot_Cyl.HomingCmd1:= TRUE;
				OP130_GVL.CR130_LH_Rot_Cyl.HomingCmd2:= FALSE;
		       END_IF
	       END_IF
	
	   90:IF (OP130_HomeRunning AND OP130_HMI_Homing)THEN  
			   SR130_LH_Servo_Control.position := 0.0;
			   SR130_LH_Servo_Control.Velocity := 10;
		       OP130_Homing_Seq:=100;
	      END_IF
	
	100:IF (OP130_HomeRunning AND OP130_HMI_Homing)THEN 
       		
			SR130_LH_Servo_Control.ABSmove_Start := TRUE;
			OP130_Homing_Seq:=115;
			END_IF
			
	115:IF SR130_LH_Servo_Control.Axis_In_Pos THEN
		  
		   SR130_LH_Servo_Control.ABSmove_Start := FALSE;
		   SR130_Stepper_Control.Bsethome := TRUE;
			IF SR130_Clm_Stepper.bHomeDone AND SR130_Clm_Stepper.baxis_in_home_pos THEN
			    OP130_Homing_Seq:=116;
            END_IF
		END_IF
	
    116: IF OP130_LH_HomeOK AND OP130_RH_HomeOK THEN
		    OP130_Homing_Seq:=120;
	     END_IF

	120: OP130_HomeRunning:=FALSE;
		 OP130_Homing_Seq:=0;
		
	
END_CASE





IF NOT OP130_HomeRunning THEN
	
	OP130_GVL.CR130_LH_Rot_Cyl.HomingCmd1:= FALSE;
	OP130_GVL.CR130_LH_Rot_Cyl.HomingCmd2:= FALSE;
	OP130_GVL.CR130_RH_Rot_Cyl.HomingCmd1:= FALSE;
	OP130_GVL.CR130_RH_Rot_Cyl.HomingCmd2:= FALSE;
				
END_IF

END_PROGRAM

// ---- POUs/Programs/OP130/OP130_RH_Initialization_Seq.TcPOU
PROGRAM OP130_RH_Initialization_Seq
VAR
END_VAR





CASE OP130_RH_Homing_Seq OF 
	
       	0: IF (OP130_Auto AND NOT OP130_HomeRunning AND  NOT OP130_ErrorActive AND  NOT OP130_AutoRunning AND NOT OP130_StepRunning	 AND NOT OP130_Temp_Home_OK) THEN
       		  OP130_HomeRunning:=TRUE;
       		  OP130_RH_Homing_Seq:=10;	
       	   END_IF
	   
	    10:IF SR130_stManualModeAxis_RH_Vert_Servo.actualPosition >=61  THEN
		      OP130_RH_Homing_Seq:=20;
	        ELSE
		      OP130_RH_Homing_Seq:=90;
		    END_IF
	   
	   20: IF (OP130_HomeRunning AND OP130_HMI_Homing)THEN 
		     // OP130_GVL.SR130_RH_Vert_Servo.fTargetPosition:=SR130_HMI_Servo_CylWork_Position;
		    // OP130_GVL.SR130_RH_Vert_Servo.fTargetVelocity:=SR130_HMI_Servo_CylWork_Velocity;
		      SR130_RH_Servo_Control.Position:=SR130_HMI_Servo_CylWork_Position;
			  SR130_RH_Servo_Control.Velocity:=SR130_HMI_Servo_CylWork_Velocity;
		      OP130_RH_Homing_Seq:=30;
	       END_IF
	   
	   30: IF (OP130_HomeRunning AND OP130_HMI_Homing)THEN 
		   //  SR130_RH_Abs_Move_Start:=TRUE;
			 SR130_RH_Servo_Control.ABSmove_Start:=TRUE;
			 OP130_RH_Homing_Seq:=40;
	       END_IF
		   
	   40:IF (OP130_HomeRunning AND OP130_HMI_Homing)THEN 
		     IF OP130_GVL.SR130_RH_Servo_Control.Axis_In_Pos THEN
			// SR130_RH_Abs_Move_Start:=FALSE;
			    SR130_RH_Servo_Control.ABSmove_Start:=FALSE;
			    OP130_RH_Homing_Seq:=50;
		     END_IF
	      END_IF
		  
	   50:IF (OP130_HomeRunning AND OP130_HMI_Homing)THEN 
		   IF CR130_RH_Rot_Cyl.Position2 THEN
			   OP130_RH_Homing_Seq:=60; 
		    ELSE
		      OP130_GVL.CR130_RH_Rot_Cyl.HomingCmd2:= TRUE;
		      OP130_GVL.CR130_RH_Rot_Cyl.HomingCmd1:= FALSE;
	       END_IF
	   END_IF
	   
	   60:IF (OP130_HomeRunning AND OP130_HMI_Homing)THEN 
		    //OP130_GVL.SR130_RH_Vert_Servo.fTargetPosition:=SR130_HMI_Servo_Rotation_Position;
		    //OP130_GVL.SR130_RH_Vert_Servo.fTargetVelocity:=SR130_HMI_Servo_Rotation_Velocity;
		     SR130_RH_Servo_Control.Position:=SR130_HMI_Servo_Rotation_Position;
		     SR130_RH_Servo_Control.Velocity:=SR130_HMI_Servo_Rotation_Velocity;
		     OP130_RH_Homing_Seq:=70;
	      END_IF
	   
	   70: IF (OP130_HomeRunning AND OP130_HMI_Homing)THEN 
		     //SR130_RH_Abs_Move_Start:=TRUE;
			   SR130_RH_Servo_Control.ABSmove_Start:=TRUE;
			   IF  OP130_GVL.SR130_RH_Servo_Control.Axis_In_Pos THEN
				 // SR130_RH_Abs_Move_Start:=FALSE;
				  SR130_RH_Servo_Control.ABSmove_Start:=FALSE;
				  OP130_RH_Homing_Seq:=80;
			   END_IF
	       END_IF
		   
	80:IF (OP130_HomeRunning AND OP130_HMI_Homing)THEN 
		  IF OP130_GVL.CR130_RH_Rot_Cyl.Position1 THEN
			OP130_RH_Homing_Seq:=90;
		  ELSE
				OP130_GVL.CR130_RH_Rot_Cyl.HomingCmd1:= TRUE;
				OP130_GVL.CR130_RH_Rot_Cyl.HomingCmd2:= FALSE;
		  END_IF
	   END_IF
	
	90:IF (OP130_HomeRunning AND OP130_HMI_Homing)THEN  
		//  OP130_GVL.SR130_RH_Vert_Servo.fTargetPosition:=0.0;
		//  OP130_GVL.SR130_RH_Vert_Servo.fTargetVelocity:=10;
		  SR130_RH_Servo_Control.Position :=0.0;
		  SR130_RH_Servo_Control.Velocity :=10;
		  OP130_RH_Homing_Seq:=100;
	   END_IF
	
	100:IF (OP130_HomeRunning AND OP130_HMI_Homing)THEN 
           SR130_RH_Abs_Move_Start:=TRUE;
	       SR130_RH_Servo_Control.ABSmove_Start:=TRUE;
			IF SR130_RH_Servo_Control.Axis_In_Pos THEN
			//   SR130_RH_Abs_Move_Start:=FALSE;
			   SR130_RH_Servo_Control.ABSmove_Start:=FALSE;
			   OP130_RH_Homing_Seq:=110;
			END_IF
		END_IF
		
	110: 
		OP130_HomeRunning:=FALSE;
		OP130_RH_Homing_Seq:=0;
	
END_CASE

END_PROGRAM

// ---- POUs/Programs/OP130/op130_tool_change.TcPOU
PROGRAM op130_tool_change
VAR
	op130_1_tool_change : tool_changeover;
	op130_2_tool_change : tool_changeover;
	fb_reset_1       :BOOL;
	fb_reset_2       :BOOL;
	
	// VERTICAL 1
	OP130_V1_TOL_UNLOD_STRT					: BOOL;
	OP130_V1_TOL_LOAD_STRT					: BOOL;
	OP130_V1_TOL_DISENGAGE					: BOOL;
	OP130_V1_TOL_ENGAGE						: BOOL;
	op130_t1_manual_lock                    : BOOL;
	op130_t1_manual_unlock                  : BOOL;
	OP130_V1_UNLD_STUS                      : STRING;
	OP130_V1_LOAD_STUS                      : STRING;
	
	// VERTICAL 2
	
	OP130_V2_TOL_UNLOD_STRT					: BOOL;
	OP130_V2_TOL_LOAD_STRT					: BOOL;
	OP130_V2_TOL_DISENGAGE					: BOOL;
	OP130_V2_TOL_ENGAGE						: BOOL;
	op130_t2_manual_lock                    : BOOL;
	op130_t2_manual_unlock                  : BOOL;
	OP130_V2_UNLD_STUS                      : STRING;
	OP130_V2_LOAD_STUS                      : STRING;
	
	tool_6_fb: BOOL;
	tool_8_fb: BOOL;
	
	OP130_TOOL_CHANGE_MODE_SELECTED: BOOL;
END_VAR


VAR PERSISTENT
	
	OP130_V1_TOL_WRK_POS					: LREAL;
	OP130_V1_TOL_HME_POS					: LREAL;
	op130_v1_TOL_VELOCITY					: LREAL;
	OP130_V1_TOL_CHNGE_CMPLE				: BOOL;
	OP130_V1_TOL_LOAD_COMPLE                : BOOL;
	OP130_V1_TOL_UNLOAD_COMPLE              : BOOL;
	   
	OP130_V2_TOL_WRK_POS					: LREAL;
	OP130_V2_TOL_HME_POS					: LREAL;
	op130_V2_T0L_VELOCITY					: LREAL;
	OP130_V2_TOL_CHNGE_CMPLE				: BOOL;
	OP130_V2_TOL_LOAD_COMPLE                : BOOL;
	OP130_V2_TOL_UNLOAD_COMPLE              : BOOL;
	
END_VAR

IF OP130_TOOL_CHANGE_MODE_SELECTED THEN
op130_1_tool_change(
	actual_pos:= , 
	actual_vel:= , 
	target_work_pos:= OP130_V1_TOL_WRK_POS, 
	target_home_pos:= OP130_V1_TOL_HME_POS, 
	target_vel_from_hmi:= op130_v1_TOL_VELOCITY, 
	station_number:= , 
	mover_number:= , 
	no_of_mover_present:= , 
	model_selected:= model_selected, 
	tool_unloading_start:=OP130_V1_TOL_UNLOD_STRT , 
	tool_loading_start:=OP130_V1_TOL_LOAD_STRT , 
	error_active:=OP130_ErrorActive , 
	station_in_auto:= OP130_Auto, 
	station_in_home:=  OP130_Temp_Home_Ok, 
	absoulte_move_done:= , 
	tool_6_3_present:= tool_6_fb, 
	tool_7_89_present:= tool_8_fb, 
	fb_reset:=fb_reset_1,
	SERVO_TOL_CHECK_OFFSET_POS := 18, 
	tool_changer_over_complete=> OP130_V1_TOL_CHNGE_CMPLE,
	tool_disengage=> OP130_V1_TOL_DISENGAGE, 
	tool_engagae=> OP130_V1_TOL_ENGAGE, 
	tool_loading_complete=> OP130_V1_TOL_LOAD_COMPLE, 
	tool_unloading_complete=> OP130_V1_TOL_UNLOAD_COMPLE, 
	servo_move_abs=>, 
	unloading_status=>OP130_V1_UNLD_STUS , 
	loading_status=>OP130_V1_LOAD_STUS,
    tool_loading_failed :=  , 
	target_pos_to_servo=> , 
	target_vel_to_servo=> );
	
	op130_2_tool_change(
	actual_pos:=  , 
	actual_vel:= , 
	target_work_pos:= OP130_V2_TOL_WRK_POS, 
	target_home_pos:= OP130_V2_TOL_HME_POS, 
	target_vel_from_hmi:= op130_V2_T0L_VELOCITY, 
	station_number:= , 
	mover_number:= , 
	no_of_mover_present:= , 
	model_selected:= model_selected, 
	tool_unloading_start:=OP130_V2_TOL_UNLOD_STRT , 
	tool_loading_start:=OP130_V2_TOL_LOAD_STRT , 
	error_active:=OP130_ErrorActive , 
	station_in_auto:= OP130_Auto, 
	station_in_home:=  OP130_Temp_Home_Ok, 
	absoulte_move_done:= SR140_Vert_Servo_Ctrl_2.Axis_In_Pos, 
	tool_6_3_present:= tool_6_fb, 
	tool_7_89_present:= tool_8_fb, 
	fb_reset:=fb_reset_1,
	SERVO_TOL_CHECK_OFFSET_POS := 18, 
	tool_changer_over_complete=> OP130_V2_TOL_CHNGE_CMPLE,
	tool_disengage=> OP130_V2_TOL_DISENGAGE, 
	tool_engagae=> OP130_V2_TOL_ENGAGE, 
	tool_loading_complete=> OP130_V2_TOL_LOAD_COMPLE, 
	tool_unloading_complete=> OP130_V2_TOL_UNLOAD_COMPLE, 
	servo_move_abs=>, 
	unloading_status=>OP130_V2_UNLD_STUS , 
	loading_status=>OP130_V2_LOAD_STUS,
    tool_loading_failed :=  , 
	target_pos_to_servo=> , 
	target_vel_to_servo=> );
	
	END_IF
	
//// op 130 tool 1 outputs/////

	
IF op130_t1_manual_lock OR OP130_V1_TOL_ENGAGE THEN
	O130_LH_TOOL_CHO_LOCK_Q1340_5     :=TRUE;
ELSIF op130_t1_manual_unlock OR OP130_V1_TOL_DISENGAGE THEN
	O130_LH_TOOL_CHO_UNLOCK_Q1340_4   :=TRUE;
ELSE
	O130_LH_TOOL_CHO_LOCK_Q1340_5     :=FALSE;
	O130_LH_TOOL_CHO_UNLOCK_Q1340_4   :=FALSE;
END_IF
   

//// op 130 tool 2 outputs///// 	

IF op130_t2_manual_lock OR OP130_V2_TOL_ENGAGE THEN
	O130_RH_TOOL_CHO_LOCK_Q1340_7      :=TRUE;
ELSIF op130_t2_manual_unlock OR OP130_V2_TOL_DISENGAGE THEN
	O130_RH_TOOL_CHO_UNLOCK_Q1340_6    :=TRUE;
ELSE
	O130_RH_TOOL_CHO_UNLOCK_Q1340_6   :=FALSE;
	O130_RH_TOOL_CHO_LOCK_Q1340_7     :=FALSE;
END_IF

END_PROGRAM

// ---- POUs/Programs/OP140/OP140_Main.TcPOU
PROGRAM OP140_Main
VAR
	OP140_ModeSelection_FB: Mode_Selection_Block1;
	//OP140_Leak_1: OP140_LeakTesting;
END_VAR

//MOdeselection From HMI
OP140_AutoSequence_1();
OP140_AutoSequence_2();
OP140_AutoSequence_3();
OP140_Error();
OP140_Manual();
Ateq_Comm_Prog();
OP140_Initialization_Seq();
op140_tool_change(); 
op140_ateq_fb();


IF (OP140_HMI_AutoMode AND NOT OP140_HMI_ManualMOde AND NOT OP140_HMI_StepMode) THEN
	OP140_Modeselection_FB.ModeWord:=1;
	ELSIF (NOT OP140_HMI_AutoMode AND OP140_HMI_ManualMOde AND NOT OP140_HMI_StepMode) THEN
		OP140_Modeselection_FB.ModeWord:=2;
	ELSIF  (NOT OP140_HMI_AutoMode AND NOT OP140_HMI_ManualMOde AND  OP140_HMI_StepMode) THEN
		OP140_Modeselection_FB.ModeWord:=3;
    ELSE   
		OP140_Modeselection_FB.ModeWord:=0;
END_IF



OP140_ModeSelection_FB(
	ModeWord:= , 
	HomeConditionOK:=OP140_HomeConditionOK , 
	OperationEnable:= OperationEnable, 
	StartPB:=OP140_HMI_CycleStart , 
	SafetyAndNOError:=OperationEnable , 
	ModeAck:=TRUE , 
	HomingINProgress:= , 
	TempHomeOK:=OP140_Temp_Home_Ok , 
	ResetPB:=OP140_HMI_Reset	 , 
	AutoSelected=>OP140_AutoSelected , 
	ManualSelected=>OP140_ManualSelected , 
	StepSelected=>OP140_StepSelected , 
	ModeSelAck_Indication=> , 
	StatusDisplay=> , 
	AutoRunning:=OP140_AutoRunning , 
	StepRunning:= OP140_StepRunning, 
	StartEnable:=OP140_StartEnable , 
	MachineStop:=OP140_Machine_Stop );
	
	IF OP140_AutoSelected THEN
		OP140_Auto:=TRUE;
		ELSE
			OP140_Auto:=FALSE;
		END_IF
		
	IF 	OP140_StartEnable THEN 
		op140_startenable_1 :=TRUE;
		op140_startenable_2 :=TRUE;
		op140_startenable_3 :=TRUE;
	ELSE
		op140_startenable_1 :=FALSE;
		op140_startenable_2 :=FALSE;
		op140_startenable_3 :=false;
	END_IF

// temp need to be deleted
//IF OP140_STN_ENABLE_1 THEN
//	OP140_STN_ENABLE_2:=TRUE;
//	OP140_STN_ENABLE_3:=TRUE;
//END_IF

END_PROGRAM

// ---- POUs/Programs/OP140/OP140_AutoSequence_1.TcPOU
PROGRAM OP140_AutoSequence_1
VAR
	OP140_STN_MOVER_1: INT;
	OP140_AutoSeq_1:INT;
	Leak1_FB: OP140_LeakTesting;
	LK1_TS1_Seq_Start: BOOL;
	LK1_TS1_Seq_Completed: BOOL;
	LK1_TS1_tst1_OK: BOOL;
	LK1_TS1_tst1_NOK: BOOL;
	LK1_TS1_tst2_OK: BOOL;
	LK1_TS1_tst2_NOK: BOOL;
	LK1_TS1_tst1_Result: STRING;
	LK1_TS1_tst2_Result: STRING;
	LK1_TS1_CompOK: BOOL;
	LK1_TS1_CompNOK: BOOL;
	LK1_TS2_Seq_Start: BOOL;
	LK1_TS2_Seq_Completed: BOOL;
	LK1_TS2_tst1_OK: BOOL;
	LK1_TS2_tst1_NOK: BOOL;
	LK1_TS2_tst2_OK: BOOL;
	LK1_TS2_tst2_NOK: BOOL;
	LK1_TS2_tst1_Result: STRING;
	LK1_TS2_tst2_Result: STRING;
	LK1_TS2_CompOK: BOOL;
	LK1_TS2_CompNOK: BOOL;
	OP140_Leak1_TS2_result_OK: BOOL;
	OP140_Leak1_TS2_result_NOK: BOOL;
	OP140_Leak1_TS2_Result_Data: STRING;
	OP140_DoneDly_1 : TON;
	OP140_STN_MOVER_1_1: INT;
	OP140_RH_AutoSeq_1: INT;
	CR140_Horz_Cyl_: INT;
	fix_lh_1: INT ;
	fix_rh_1:INT;
	Dry_run : BOOL;
	DON_FAL_TRG: F_TRIG;
END_VAR

 VAR
	 OP140_Leak1_TS1_result_OK:BOOL;
	OP140_Leak1_TS1_Result_NOK:BOOL;
	OP140_Leak1_TS1_Result_Data:STRING;
	OP1140_LK1_LH_OK:BOOL;
	OP1140_LK1_LH_NOK:BOOL;
	OP1140_LK1_RH_OK:BOOL;
	OP1140_LK1_RH_NOK:BOOL;
	op140_step_time_fb :step_cycle_time;
	op140_step_no      :ARRAY [1..20] OF INT;
	op140_step_time    :ARRAY [1..20] OF UDINT;
	
 END_VAR

IF (NOT OP140_Auto OR  OP140_ErrorActive OR OP140_HomeRunning OR OP140_Machine_Stop ) THEN
	
// used in sequence	 all auto as seperate bits
    OP140_ComponentOk:=FALSE;
    OP140_ComponentNok:=FALSE;
	OP140_Leak1_Seq_Completed:=FALSE;
	OP140_Leak1_Seq_Start:=FALSE;
	OP140A1_Prev_LH_COMP_OK:=FALSE;
	OP140A1_Prev_RH_COMP_OK:=FALSE;
	OP140_AutoSeq_1:= 10;
	OP140_AutoRunning:= FALSE;
	OP140_ATEQ6_ResultOK :=FALSE;
	OP140_ATEQ6_ResultNOK :=FALSE;
	OP140_ATEQ3_ResultOK :=FALSE;
	OP140_ATEQ3_ResultNOK :=FALSE;
	
END_IF

CASE OP140_AutoSeq_1 OF 
	
	10:IF (OP140_Auto) THEN		// Check Automode Selected
		  OP140_AutoSeq_1 :=20;
	   END_IF
	   
	20:IF ( NOT OP140_ErrorActive) THEN		//Check No error
		OP140_AutoSeq_1:=30;
	   END_IF
	   
	30:IF (NOT OP140_HomeRunning) THEN		//Check No Homerunning
		OP140_AutoSeq_1 :=40;
		END_IF
		
    40:IF ( OP140_Temp_Home_Ok)THEN	//Check Machine in Home
		OP140_AutoSeq_1:= 50;
		END_IF
		
	50:IF ( NOT OP140_OperationCompleted) AND NOT OP140_TOOL_CHANGE_MODE_SELECTED THEN		// Check Operation Completed Reset
		OP140_AutoSeq_1:=60;
		END_IF
		
	60:IF (NOT OP140_ComponentOk) THEN		// Check Component Ok Reset
		OP140_AutoSeq_1:=70;
		END_IF
		
	70:IF (NOT OP140_ComponentNok) THEN 	// Check Component NOk Reset
		OP140_AutoSeq_1:= 120;
		END_IF
		
    120:IF  ( OP140_HMI_Cycle_Start ) THEN		//Machine Start in Fully Automatic or Press Cycle Start For Semi Automatic
		    OP140_HomeConditionOK:=TRUE;
	 		IF( OP140_HomeConditionOK AND OP140_AutoSelected) THEN
			   OP140_AutoRunning:=TRUE;
			   OP140_StepRunning:= FALSE;
			ELSIF ( OP140_HomeConditionOK AND OP140_StepSelected) THEN
				  OP140_AutoRunning:=FALSE;
				  OP140_StepRunning:= TRUE;
			END_IF;
		 END_IF
		 
		 IF ((OP140_AutoRunning OR OP140_StepRunning) AND OP140_StartEnable_1)AND  (OP140_DryRun OR OP140_HMI_Cycle_Start)   THEN
              OP140_AutoSeq_1:= 130;
		END_IF
		
	130:IF  OP140_STN_ENABLE_1  THEN 
 			OP140_AutoSeq_1:= 140;
			
		ELSIF NOT  OP140_STN_ENABLE_1 AND MOVER_POS_RECHED[OP140_STN_MOVER_1] AND
		           fix_lh_1 <> 130 AND fix_rh_1 <> 130 THEN
		           OP140_AutoSeq_1 := 200;
		END_IF
		
	140:IF fix_lh_1 =130 AND fix_rh_1 =130 THEN
		   OP140A1_Prev_LH_COMP_OK := TRUE;
	       OP140A1_Prev_RH_COMP_OK := TRUE;
   		   OP140_AutoSeq_1 := 150;																																																																																				
		ELSIF fix_lh_1 =130 AND fix_rh_1 =131 THEN
			  OP140A1_Prev_LH_COMP_OK := TRUE;
	          OP140A1_Prev_RH_COMP_OK := FALSE;
			  OP140_AutoSeq_1 := 150;
		ELSIF fix_lh_1 =131 AND fix_rh_1 =130 THEN
			  OP140A1_Prev_LH_COMP_OK := FALSE;
	          OP140A1_Prev_RH_COMP_OK :=TRUE ;
	          OP140_AutoSeq_1 := 150;
		END_IF
			
		   

			
	150:IF OP140_StartEnable_1  THEN
		 OP140_Leak1_Seq_Start:=TRUE;	
		 OP140_AutoSeq_1:= 160;
		END_IF
		 
		 
	160:IF OP140_Leak1_Seq_Completed=TRUE AND In_Range(SR140_Vert_Servo_Ctrl_1.Actual_Position,40,1)  THEN
		  OP140A1_LH_Comp_OK:=OP1140_LK1_LH_OK;
		  OP140A1_LH_Comp_NOK:=OP1140_LK1_LH_NOK;
		  OP140A1_RH_Comp_OK:=OP1140_LK1_RH_OK;
		  OP140A1_RH_Comp_NOK:=OP1140_LK1_RH_NOK;
		IF ((Componenets_Produced MOD 100)=0 AND (Componenets_Produced > 1)) THEN
		  OP140_AutoSeq_1:= 161;
        ELSE OP140_AutoSeq_1:= 170;		
	    END_IF
		END_IF
		OP140_P1_CURR_MVR			:= OP140_STN_MOVER_1;
		
	161 : OP140_AutoSeq_1:= 170;
		
		
	170: IF OP140_DoneDly_1.q AND OP140_StartEnable THEN
		    IF OP140A1_LH_Comp_OK AND OP140A1_RH_Comp_OK THEN
		       MOVER_CMP_STATUS[OP140_P1_CURR_MVR][1]:=140;
		       MOVER_CMP_STATUS[OP140_P1_CURR_MVR][2]:=140;	

		       IF MOVER_CMP_STATUS[OP140_P1_CURR_MVR][1]=140 AND MOVER_CMP_STATUS[OP140_P1_CURR_MVR][2]=140 THEN
				STATION_DONE[OP140_P1_CURR_MVR][OP140_XTS_POS_NO]			:= TRUE;
				  OP140_AutoSeq_1:= 180;
		       END_IF 	
				
             ELSIF OP140A1_LH_Comp_NOK AND OP140A1_RH_Comp_NOK  THEN
				   MOVER_CMP_STATUS[OP140_P1_CURR_MVR][1]:=141;
		           MOVER_CMP_STATUS[OP140_P1_CURR_MVR][2]:=141;

		          IF MOVER_CMP_STATUS[OP140_P1_CURR_MVR][1]=141 AND MOVER_CMP_STATUS[OP140_P1_CURR_MVR][2]=141 THEN
				STATION_DONE[OP140_P1_CURR_MVR][OP140_XTS_POS_NO]			:= TRUE;
				     OP140_AutoSeq_1:= 180;
		          END_IF 
				
             ELSIF OP140A1_LH_Comp_OK AND OP140A1_RH_Comp_NOK  THEN
				 MOVER_CMP_STATUS[OP140_P1_CURR_MVR][1]:=140;
		         MOVER_CMP_STATUS[OP140_P1_CURR_MVR][2]:=141;
				 
		         IF MOVER_CMP_STATUS[OP140_P1_CURR_MVR][1]=140 AND MOVER_CMP_STATUS[OP140_P1_CURR_MVR][2]=141 THEN
				STATION_DONE[OP140_P1_CURR_MVR][OP140_XTS_POS_NO]			:= TRUE;
				    OP140_AutoSeq_1:= 180;
		        END_IF 	
				
			ELSIF OP140A1_LH_Comp_NOK AND OP140A1_RH_Comp_OK  THEN
				  MOVER_CMP_STATUS[OP140_P1_CURR_MVR][1]:=141;
		          MOVER_CMP_STATUS[OP140_P1_CURR_MVR][2]:=140;

		         IF MOVER_CMP_STATUS[OP140_P1_CURR_MVR][1]=141 AND MOVER_CMP_STATUS[OP140_P1_CURR_MVR][2]=140 THEN
				STATION_DONE[OP140_P1_CURR_MVR][OP140_XTS_POS_NO]			:= TRUE;
				    OP140_AutoSeq_1:= 180;
		        END_IF 		
		    END_IF		
	     END_IF
	
	180:// Reset All Bits
		OP140_Leak1_Seq_Completed:=FALSE;					
        OP140A1_LH_Comp_OK       :=FALSE;
        OP140A1_LH_Comp_NOK      :=FALSE;
        OP140A1_RH_Comp_OK       :=FALSE;
        OP140A1_RH_Comp_NOK      :=FALSE;
        OP140_ATEQ6_ResultOK     :=FALSE;
		OP140_ATEQ6_ResultNOK    :=FALSE;
		OP140_ATEQ3_ResultOK     :=FALSE;
		OP140_ATEQ3_ResultNOK    :=FALSE;
		OP140_STN_ENABLE_1       :=0;
		OP140_AutoSeq_1          := 130;	


	200:/// all sequence skip	
        MOVER_CMP_STATUS[OP140_P1_CURR_MVR][2]:=141;
		MOVER_CMP_STATUS[OP140_P1_CURR_MVR][1]:=141;		
		IF MOVER_CMP_STATUS[OP140_P1_CURR_MVR][1]=141 AND MOVER_CMP_STATUS[OP140_P1_CURR_MVR][2]=141 THEN
		STATION_DONE[OP140_STN_MOVER_1][OP140_XTS_POS_NO]			:= TRUE;
				OP140_AutoSeq_1:= 180;
		END_IF		

END_CASE



Leak1_FB(
	
	Horz_Cyl_Pos1            := CR140_Horz_Cyl_1.Position1, 
	Horz_Cyl_Pos2            :=CR140_Horz_Cyl_1.Position2 , 
	Vert_Cyl_Pos1            := CR140_Vert_Cyl_1.Position1, 
	Vert_Cyl_Pos2            := CR140_Vert_Cyl_1.Position2, 
	StartEnable              :=OP140_StartEnable_1 , 
	Home_pos_IP              :=OP140_HMI_Vert_Home_Pos, 
	Home_Vel_IP              := OP140_HMI_Vert_Home_Vel,
	SafeHome_Pos_IP          :=OP140_HMI_Vert_SafeHome_Pos,
	SafeHome_Vel_Ip          :=OP140_HMI_Vert_SafeHome_Vel, 
	SafeWork_Pos_IP          :=OP140_HMI_Vert_SafeWork_Pos,
	SafeWork_Vel_IP          :=OP140_HMI_Vert1_SafeWork_Vel,
	Work_Pos_IP              :=OP140_HMI_Vert1_Work_Pos , 
	Work_Vel_IP              :=OP140_HMI_Vert1_Work_Vel , 
	Axis_In_WorkPos          :=SR140_Vert_Servo_Ctrl_1.Axis_In_Pos , 
	Axis_In_Home             :=SR140_Vert_Servo_Ctrl_1.Axis_In_Home , 
	axis_in_position         :=SR140_Vert_Servo_Ctrl_1.Axis_In_Pos,
	servo_actual_pos         :=SR140_Vert_Servo_Ctrl_1.Actual_Position,
	Prev_Stat_LH_OK          :=OP140A1_Prev_LH_COMP_OK , 
	Prev_Stat_RH_OK          :=OP140A1_Prev_RH_COMP_OK , 
	TS1_Test1_ProgNO         :=OP140_ATEQ_Test_Prog1_No , 
	TS1_Test2_ProgNO         :=OP140_ATEQ_Test_Prog2_No , 
	TS1_TestOk               :=OP140_ATEQ6_ResultOK , 
	TS1_TestNOK              :=OP140_ATEQ6_ResultNOK , 
	TS1_StartEnable          := OP140_StartEnable_1, 
	TS1_ResultIN             := OP140_ATEQ6_Result , 
	TS2_Test1_ProgNO         :=OP140_ATEQ_Test_Prog1_No , 
	TS2_Test2_ProgNO         :=OP140_ATEQ_Test_Prog2_No , 
	TS2_TestOk               :=OP140_ATEQ3_ResultOK , 
	TS2_TestNOK              :=OP140_ATEQ3_ResultNOK , 
	TS2_StartEnable          :=OP140_StartEnable_1 , 
	TS2_ResultIN             :=OP140_ATEQ3_Result , 
	Horz_Cyl_Auto1           =>CR140_Horz_Cyl_1.AutoCmd1 , 
	Horz_Cyl_Auto2           =>CR140_Horz_Cyl_1.AutoCmd2 , 
	Vert_Cyl_Auto1           =>CR140_Vert_Cyl_1.AutoCmd1 , 
	Vert_Cyl_Auto2           =>CR140_Vert_Cyl_1.AutoCmd2 , 
	Servo_Pos_Error          => , 
	Servo_HomePos_Error      => , 
	TS1_StartOP              => OP140_ATEQ6_Auto_Start , 
	TS1_Test_ProgNO          => OP140_ATEQ6_Auto_Prog_No_out , 
	TS2_StartOP              =>OP140_ATEQ3_Auto_Start , 
	TS2_Test_ProgNO          => OP140_ATEQ3_Auto_Prog_No_out , 
	Seq_Start                := OP140_Leak1_Seq_Start, 
	Seq_Completed            :=OP140_Leak1_Seq_Completed , 
	TS1_SeqStart             :=LK1_TS1_Seq_Start , 
	TS1_SeqCompleted         := LK1_TS1_Seq_Completed, 
	TS1_ATEQCompleted        :=  OP140_ATEQ6_ResultCompleted, 
	TS1_Test1OK              :=LK1_TS1_tst1_OK , 
	TS1_Test1NOK             := LK1_TS1_tst1_NOK, 
	TS1_Test2Ok              :=LK1_TS1_tst2_OK , 
	TS1_Test2NOK             :=LK1_TS1_tst2_NOK , 
	TS1_Test1Result          := LK1_TS1_tst1_Result, 
	TS1_Test2Result          :=LK1_TS1_tst2_Result , 
	TS1_CompOK               :=LK1_TS1_CompOK , 
	TS1_CompNOK              := LK1_TS1_CompNOK, 
	TS1_ResultOK             :=OP140_Leak1_TS1_result_OK , 
	TS1_ResultNOK            := OP140_Leak1_TS1_Result_NOK, 
	TS1_Result_Data          :=OP140_Leak1_TS1_Result_Data , 
	LH_CompOK                :=OP1140_LK1_LH_OK , 
	LH_CompNOK               :=OP1140_LK1_LH_NOK , 
	RH_CompOK                :=OP1140_LK1_RH_OK , 
	RH_CompNOK               :=OP1140_LK1_RH_NOK , 
	TS2_SeqStart             :=LK1_TS2_Seq_Start , 
	TS2_SeqCompleted         := LK1_TS2_Seq_Completed , 
	TS2_ATEQCompleted        :=OP140_ATEQ3_ResultCompleted , 
	TS2_Test1OK              :=LK1_TS2_tst1_OK , 
	TS2_Test1NOK             :=LK1_TS2_tst1_NOK  , 
	TS2_Test2Ok              :=LK1_TS2_tst2_OK , 
	TS2_Test2NOK             :=LK1_TS2_tst2_NOK , 
	TS2_Test1Result          := LK1_TS2_tst1_Result , 
	TS2_Test2Result          :=LK1_TS2_tst2_Result , 
	TS2_CompOK               :=LK1_TS2_CompOK , 
	TS2_CompNOK              :=LK1_TS2_CompNOK , 
	TS2_ResultOK             := OP140_Leak1_TS2_result_OK, 
	TS2_ResultNOK            :=OP140_Leak1_TS2_result_NOK , 
	TS2_Result_Data          :=OP140_Leak1_TS2_Result_Data ,
    Servo_Pos_OP             :=SR140_Vert_Servo_Ctrl_1.Position,
    Servo_Vel_OP             :=SR140_Vert_Servo_Ctrl_1.Velocity,
    ABS_Move_Start           :=SR140_Vert_Servo_Ctrl_1.ABSmove_Start);

// cycle time
op140_step_time_fb(step_numbers:= op140_step_no, auto_step_no:=OP140_AutoSeq_1 , step_time=>op140_step_time );
OP140_DoneDly_1(IN:=OP140_Leak1_Seq_Completed , PT:=T#500MS , Q=> , ET=> );
dry_run:=All_Station_Dry_Run;	
IF Dry_Run THEN
	fix_lh_1:=130;	
    fix_rh_1:=130;
ELSE
	fix_lh_1:=MOVER_CMP_STATUS[OP140_STN_MOVER_1][1];	
    fix_rh_1:=MOVER_CMP_STATUS[OP140_STN_MOVER_1][2];	
END_IF

//############################		OP140 STATION ENABLE CONDITION		##########################

	OP140_STN_MOVER_1					:= MOVER_POSITION[OP140_P1_XTS_POS_NO];
	
	IF AUTO_WITH_XTS THEN
	IF OP140_STN_MOVER_1>0 THEN	
	IF NOT(END_OF_CYCLE AND MOVER_CMP_STATUS[OP140_STN_MOVER_1][1]=5 AND MOVER_CMP_STATUS[OP140_STN_MOVER_1][2]=5)THEN
	OP140_STN_ENABLE_1					:= MOVER_POS_RECHED[OP140_STN_MOVER_1] AND ((MOVER_CMP_STATUS[OP140_STN_MOVER_1][1]=130)OR 
										(MOVER_CMP_STATUS[OP140_STN_MOVER_1][2]=130))AND STATION_ENABLE_CONTROL;	
	ELSE
	STATION_DONE[OP140_STN_MOVER_1][OP140_XTS_POS_NO]			:= TRUE;		
	END_IF
	ELSE
	OP140_STN_ENABLE_1					:= FALSE;	
	END_IF
	END_IF

END_PROGRAM

// ---- FB/OP140_LeakTesting.TcPOU
FUNCTION_BLOCK OP140_LeakTesting
VAR_INPUT
	Horz_Cyl_Pos1:BOOL;
	Horz_Cyl_Pos2:BOOL;
	Vert_Cyl_Pos1:BOOL;
	Vert_Cyl_Pos2:BOOL;
	StartEnable:BOOL;
	Home_pos_IP:LREAL;
	Home_Vel_IP:LREAL;
	SafeHome_Pos_IP:LREAL;
	SafeHome_Vel_Ip:LREAL;
	SafeWork_Pos_IP:LREAL;
	SafeWork_Vel_IP:LREAL;
	Work_Pos_IP:LREAL;
	Work_Vel_IP:LREAL;
	Axis_In_WorkPos:BOOL;
	Axis_In_Home:BOOL;
	Prev_Stat_LH_OK:BOOL;
	Prev_Stat_RH_OK:BOOL;
	servo_actual_pos:LREAL;
	axis_in_position :bool;
	//TestSeq1 I/P
	
	TS1_Test1_ProgNO:INT;
	TS1_Test2_ProgNO:INT;
	TS1_TestOk:BOOL;
	TS1_TestNOK:BOOL;
	TS1_StartEnable:BOOL;
	TS1_ResultIN:STRING;
	
	//TestSeq2 I/P
	
	TS2_Test1_ProgNO:INT;
	TS2_Test2_ProgNO:INT;
	TS2_TestOk:BOOL;
	TS2_TestNOK:BOOL;
	TS2_StartEnable:BOOL;
	TS2_ResultIN:STRING;
	
	
END_VAR
VAR_OUTPUT
	Horz_Cyl_Auto1:BOOL;
	Horz_Cyl_Auto2:BOOL;
	Vert_Cyl_Auto1:BOOL;
	Vert_Cyl_Auto2:BOOL;
	
	
	Servo_Pos_Error:BOOL;
	Servo_HomePos_Error:BOOL;
	
//TestSeq1 O/P

	TS1_StartOP:BOOL;
	TS1_Test_ProgNO:INT;
//TestSeq2 O/P

	TS2_StartOP:BOOL;
	TS2_Test_ProgNO:INT;
	actual_step_no: INT;
END_VAR
VAR_IN_OUT
	
	//LH_ATEQ_FB:ATEQ_Fb;
	//RH_ATEQ_FB:ATEQ_Fb;
	Seq_Start:BOOL;
	Seq_Completed:BOOL;
	//TestSeq INOUt
	TS1_SeqStart:BOOL;
	TS1_SeqCompleted:BOOL;
	TS1_ATEQCompleted:BOOL;
	TS1_Test1OK:BOOL;
	TS1_Test1NOK:BOOL;
	TS1_Test2Ok:BOOL;
	TS1_Test2NOK:BOOL;
	TS1_Test1Result:STRING;
	TS1_Test2Result:STRING;
	TS1_CompOK:BOOL;
	TS1_CompNOK:BOOL;
	TS1_ResultOK:BOOL;
	TS1_ResultNOK:BOOL;
	TS1_Result_Data:STRING;
	LH_CompOK:BOOL;
	LH_CompNOK:BOOL;
	RH_CompOK:BOOL;
	RH_CompNOK:BOOL;
	//TestSeq2 IN OUT
	
	TS2_SeqStart:BOOL;
	TS2_SeqCompleted:BOOL;
	TS2_ATEQCompleted:BOOL;
	TS2_Test1OK:BOOL;
	TS2_Test1NOK:BOOL;
	TS2_Test2Ok:BOOL;
	TS2_Test2NOK:BOOL;
	TS2_Test1Result:STRING;
	TS2_Test2Result:STRING;
	TS2_CompOK:BOOL;
	TS2_CompNOK:BOOL;
	TS2_ResultOK:BOOL;
	TS2_ResultNOK:BOOL;
	TS2_Result_Data:STRING;
	Servo_Pos_OP:LREAL;
	Servo_Vel_OP:LREAL;
	ABS_Move_Start:BOOL;
	
END_VAR
	

VAR
	Step_No:INT;
	LH_Operation_Inhibit:BOOL;
	RH_Operation_Inhibit:BOOL;
	Test_Count:INT;
	ServoPOsErr: TON;
	ServoHomePosErr: TON;
	TS1: TestSeq;
	TS2: TestSeq;
END_VAR

IF NOT StartEnable THEN
	Step_No:=0;
END_IF


CASE Step_No OF 
	0:Seq_Start:=FALSE;
	  Seq_Completed:=FALSE;
	  Horz_Cyl_Auto1:=FALSE;
	  Horz_Cyl_Auto2:=FALSE;
	  Vert_Cyl_Auto1:=FALSE;
			Vert_Cyl_Auto2:=FALSE;
	 
	  TS1_SeqStart:=FALSE;
	  TS2_SeqStart:=FALSE;
	  TS1_SeqCompleted:=FALSE;
	  TS2_SeqCompleted:=FALSE;
	  Step_No:=10;
	  
	  10:IF (Seq_Start= TRUE) AND (Seq_Completed=FALSE) THEN
		   Seq_Start:=FALSE;
		   Step_No:=20;
	     END_IF
		 
	  20:IF (StartEnable=TRUE) THEN
		  IF (Horz_Cyl_Pos2=TRUE) THEN 
			  Step_No:=30;
			  ELSE
				  Horz_Cyl_Auto2:=TRUE;
				  Horz_Cyl_Auto1:=FALSE;
				  IF (Horz_Cyl_Pos2=TRUE) THEN 
			       Step_No:=30;		  
		          END_IF
		      END_IF
		END_IF
		
		30:IF (StartEnable=TRUE) THEN 
			
			Vert_Cyl_Auto2:=TRUE;
			Vert_Cyl_Auto1:=FALSE;
			Servo_Pos_OP:=Work_Pos_IP;
			Servo_Vel_OP:=Work_Vel_IP;
			ABS_Move_Start:=TRUE;
			IF Axis_In_WorkPos AND Vert_Cyl_Pos2 THEN
			   ABS_Move_Start:=FALSE;
			   Step_No:=60;
			END_IF
			//IF (Vert_Cyl_Pos2=TRUE) THEN
			//	//Step_No:=40;	
			//END_IF
		END_IF
		
		40:IF (StartEnable=TRUE) THEN 
			  Servo_Pos_OP:=SafeWork_Pos_IP;
			  Servo_Vel_OP:=SafeWork_Vel_IP;
			  Step_No:=50;	
			 END_IF
			 
		50: IF (StartEnable=TRUE) THEN 
			ABS_Move_Start:=TRUE;
			IF Axis_In_WorkPos=TRUE THEN
				ABS_Move_Start:=FALSE;
				Step_No:=55;
			END_IF
		    END_IF
			
		55:	 IF (StartEnable=TRUE) THEN 
			Servo_Pos_OP:=Work_Pos_IP;
			Servo_Vel_OP:=Work_Vel_IP;
			
			ABS_Move_Start:=TRUE;
			IF Axis_In_WorkPos=TRUE THEN
				ABS_Move_Start:=FALSE;
				Step_No:=60;
			END_IF
		    END_IF
			
	   60:   IF (StartEnable=TRUE) THEN 
		
	         IF Prev_Stat_LH_OK THEN
		        TS1_SeqStart:=TRUE;
	         ELSE
		        TS1_SeqStart:=FALSE;
		        TS1_SeqCompleted:=TRUE;
		     END_IF
	         IF Prev_Stat_RH_OK THEN
		        TS2_SeqStart:=TRUE;
	         ELSE
		        TS2_SeqStart:=FALSE;
		        TS2_SeqCompleted:=TRUE;
		     END_IF
	         Step_No:=70;
		     END_IF
			 
	70:IF (StartEnable=TRUE) AND TS1_SeqCompleted AND TS2_SeqCompleted  THEN 
		
      IF TS1_ResultOK THEN
		  LH_CompOK:=TRUE;
		   LH_CompNOK:=FALSE;
	  ELSE
		  LH_CompNOK:=TRUE;
		  LH_CompOK:=TRUE;
	  END_IF
	   IF TS2_ResultOK THEN
		  RH_CompOK:=TRUE;
		  RH_CompNOK:=FALSE;
	    ELSE
		  RH_CompNOK:=TRUE;
		  RH_CompOK:=FALSE;
	    END_IF
        IF (LH_CompOK OR LH_CompNOK) AND (RH_CompOK OR RH_CompNOK) THEN
		   Step_No:=75;
	    END_IF
	    END_IF
		
	75:IF (StartEnable=TRUE)   THEN
	      TS1_SeqCompleted:=FALSE;
		  TS2_SeqCompleted:=FALSE;
		  Servo_Pos_OP:=SafeHome_Pos_IP;
		  Servo_Vel_OP:=SafeHome_Vel_Ip;
		  ABS_Move_Start:=TRUE;
		  IF  Axis_In_WorkPos THEN
			  Step_No:=80;	
			END_IF
		  END_IF
		  
		80: IF (StartEnable) THEN
			Servo_Pos_OP:=Home_pos_IP;
			Servo_Vel_OP:=Home_Vel_IP;
			ABS_Move_Start:=TRUE;
			Vert_Cyl_Auto1:=TRUE;
			Vert_Cyl_Auto2:=FALSE;
			IF (Vert_Cyl_Pos1 AND In_Range(servo_actual_pos,SafeWork_Pos_IP,1)) THEN
				Step_No:=95;
				ABS_Move_Start:=FALSE;
			END_IF
		END_IF
		95: IF (StartEnable=TRUE) THEN
		  IF (Horz_Cyl_Pos1=TRUE) THEN 
			  
		 	Seq_Completed:=TRUE;
			  Step_No:=100;
			  ELSE
				  Horz_Cyl_Auto1:=TRUE;
				  Horz_Cyl_Auto2:=FALSE;
		      END_IF
		END_IF
	
			  
 	
	100:IF NOT Seq_Completed THEN
		Seq_Completed:=FALSE;
		 LH_CompOK:=FALSE;
		   LH_CompNOK:=FALSE;
		    RH_CompNOK:=FALSE;
		  RH_CompOK:=FALSE;
		Step_NO:=0;
	    END_IF	
	
END_CASE

TS1(
	Test1_ProgNO:=TS1_Test1_ProgNO , 
	Test2_ProgNO:= TS1_Test2_ProgNO, 
	TestOk:=TS1_TestOk , 
	TestNOK:= TS1_TestNOK, 
	StartEnable:=TS1_StartEnable , 
	ResultIN:=TS1_ResultIN , 
	ATEQCompleted:=TS1_ATEQCompleted , 
	StartOP=>TS1_StartOP , 
	Test_ProgNO=>TS1_Test_ProgNO , 
	SeqStart:= TS1_SeqStart, 
	SeqCompleted:=TS1_SeqCompleted , 
	Test1OK:=TS1_Test1OK , 
	Test1NOK:=TS1_Test1NOK , 
	Test2Ok:=TS1_Test2Ok , 
	Test2NOK:=TS1_Test2NOK , 
	Test1Result:=TS1_Test1Result , 
	Test2Result:= TS1_Test2Result, 
	CompOK:= TS1_CompOK, 
	CompNOK:=TS1_CompNOK , 
	ResultOK:=TS1_ResultOK , 
	ResultNOK:= TS1_ResultNOK, 
	Result_Data:=TS1_Result_Data );
	
TS2(
	Test1_ProgNO:=TS2_Test1_ProgNO , 
	Test2_ProgNO:= TS2_Test2_ProgNO, 
	TestOk:=TS2_TestOk , 
	TestNOK:= TS2_TestNOK, 
	StartEnable:=TS2_StartEnable , 
	ResultIN:=TS2_ResultIN , 
	ATEQCompleted:=TS2_ATEQCompleted , 
	StartOP=>TS2_StartOP , 
	Test_ProgNO=>TS2_Test_ProgNO , 
	SeqStart:= TS2_SeqStart, 
	SeqCompleted:=TS2_SeqCompleted , 
	Test1OK:=TS2_Test1OK , 
	Test1NOK:=TS2_Test1NOK , 
	Test2Ok:=TS2_Test2Ok , 
	Test2NOK:=TS2_Test2NOK , 
	Test1Result:=TS2_Test1Result , 
	Test2Result:= TS2_Test2Result, 
	CompOK:= TS2_CompOK, 
	CompNOK:=TS2_CompNOK , 
	ResultOK:=TS2_ResultOK , 
	ResultNOK:= TS2_ResultNOK, 
	Result_Data:=TS2_Result_Data );









//ServoHomePosErr(IN:=Step_No:=80 , PT:=T#2S , Q=> , ET=> );
//IF Step_No=80  AND NOT Axis_In_Home AND ServoHomePosErr.q THEN
	//Servo_HomePos_Error:=TRUE;
	//END_IF
	
actual_step_no := Step_No;

END_FUNCTION_BLOCK

// ---- FB/TestSeq.TcPOU
FUNCTION_BLOCK TestSeq
VAR_INPUT
	
	Test1_ProgNO:INT;
	Test2_ProgNO:INT;
	TestOk:BOOL;
	TestNOK:BOOL;
	StartEnable:BOOL;
	ResultIN:STRING;
	
	
	
	
END_VAR
VAR_OUTPUT
	StartOP:BOOL;
	Test_ProgNO:INT;
	
	
END_VAR
VAR
	StepNO:INT;
	SeqRunning:BOOL;
	
END_VAR
VAR_IN_OUT
	SeqStart:BOOL;
	SeqCompleted:BOOL;
	Test1OK:BOOL;
	Test1NOK:BOOL;
	Test2Ok:BOOL;
	Test2NOK:BOOL;
	Test1Result:STRING;
	Test2Result:STRING;
	CompOK:BOOL;
	CompNOK:BOOL;
	ResultOK:BOOL;
	ResultNOK:BOOL;
	Result_Data:STRING;
	ATEQCompleted:BOOL;
END_VAR

IF  NOT StartEnable THEN
	StepNO:=0;
END_IF
CASE StepNO OF
	0: SeqStart:=FALSE;
	StartOP:=FALSE;
	SeqRunning:=FALSE;
	ATEQCompleted:=FALSE;
	ResultNOK:=FALSE;
	ResultOK:=FALSE;
	SeqCompleted:=FALSE;
	StepNO:=10;
	10:IF StartEnable AND SeqStart THEN
 			 			
	SeqRunning:=TRUE;
	SeqStart:=FALSE;
	StepNO:=20;
	END_IF;
20: IF StartEnable AND SeqRunning THEN
	
		Test_ProgNO:=Test1_ProgNO;
		
		StepNO:=30;
	END_IF
30: IF StartEnable AND SeqRunning THEN
	
		StartOP:=TRUE;
		StepNO:=40;
		
END_IF
40: IF ATEQCompleted AND StartEnable THEN
StartOP:=FALSE;	

	IF (TestOk AND NOT TestNOK) THEN
		ResultOK:=TRUE;
		ResultNOK:=FALSE;
	ELSIF (TestNOk AND NOT TestOK) THEN
		ResultNOK:=TRUE;
		ResultOK:=FALSE;
	END_IF
		IF (ResultOK OR ResultNOK) THEN
			StepNO:=50;
		
		END_IF
		END_IF
50: IF StartEnable THEN
	ATEQCompleted:=FALSE;
	Result_Data:=ResultIN;
	StepNO:=60;
END_IF
60:
		 IF StartEnable  THEN
			SeqCompleted:=TRUE;
			StepNO:=70;  
		 END_IF
70: IF NOT SeqCompleted THEN
		ResultNOK:=FALSE;
		ResultOK:=FALSE;
		Result_Data:='';
		StepNO:=0;
		END_IF

	
	
	
END_CASE

END_FUNCTION_BLOCK

// ---- FB/tool/step_cycle_time.TcPOU
FUNCTION_BLOCK step_cycle_time
VAR_INPUT
step_numbers            :ARRAY [1..20] OF INT ;
auto_step_no            :INT;
END_VAR

VAR_OUTPUT
step_time               : ARRAY [1..20] OF UDINT;	
END_VAR

VAR
help_var                : ARRAY [1..20] OF BOOL;
step_startTime			: ARRAY [1..20] OF ULINT;
step_time_seq           : INT:=10;
Time_diff               : ARRAY [1..20] OF UDINT;
END_VAR


(*IF step_numbers[j] <> auto_step_no THEN
		IF step_numbers[j] = auto_step_no THEN
   			help_var := TRUE;	
   			IF help_var THEN
	  			 step_startTime[j]:= F_GetSystemTime();
				 j:=j+1;
				 help_var:=0;	 
   			END_IF
		ELSE
			j:=j+1;
		END_IF
END_IF	*)

CASE step_time_seq OF

10:	IF step_numbers[1] = auto_step_no THEN
   help_var[1] := TRUE;	
   IF help_var[1] THEN
	   step_startTime[1]:= F_GetSystemTime();
	   step_time_seq:=20;
   END_IF
END_IF

20:IF step_numbers[2] = auto_step_no THEN
   help_var[2] := TRUE;	
   IF help_var[2] THEN
	   step_startTime[2]:= F_GetSystemTime();
	    step_time_seq:=30;
   END_IF
END_IF

30:IF step_numbers[3] = auto_step_no THEN
   help_var[3] := TRUE;	
   IF help_var[3] THEN
	   step_startTime[3]:= F_GetSystemTime();
	    step_time_seq:=40;
   END_IF
END_IF

40:IF step_numbers[4] = auto_step_no THEN
   help_var[4] := TRUE;	
   IF help_var[4] THEN
	   step_startTime[4]:= F_GetSystemTime();
	    step_time_seq:=50;
   END_IF
END_IF

50:IF step_numbers[5] = auto_step_no THEN
   help_var[5] := TRUE;	
   IF help_var[5] THEN
	   step_startTime[5]:= F_GetSystemTime();
	    step_time_seq:=60;
   END_IF
END_IF

60:IF step_numbers[6] = auto_step_no THEN
   help_var[6] := TRUE;	
   IF help_var[6] THEN
	   step_startTime[6]:= F_GetSystemTime();
	    step_time_seq:=70;
   END_IF
END_IF

70:IF step_numbers[7] = auto_step_no THEN
   help_var[7] := TRUE;	
   IF help_var[7] THEN
	   step_startTime[7]:= F_GetSystemTime();
	    step_time_seq:=80;
   END_IF
END_IF

80:IF step_numbers[8] = auto_step_no THEN
   help_var[8] := TRUE;	
   IF help_var[8] THEN
	   step_startTime[8]:= F_GetSystemTime();
	    step_time_seq:=90;
   END_IF
END_IF

90:IF step_numbers[9] = auto_step_no THEN
   help_var[9] := TRUE;	
   IF help_var[9] THEN
	  step_startTime[9]:= F_GetSystemTime();
	   step_time_seq:=100;
   END_IF
END_IF

100:IF step_numbers[10] = auto_step_no THEN
   help_var[10] := TRUE;	
   IF help_var[10] THEN
	   step_startTime[10]:= F_GetSystemTime();
	    step_time_seq:=200;
   END_IF
END_IF

200 :IF step_numbers[10] <> auto_step_no THEN
   help_var[11] := TRUE;	
   IF help_var[11] THEN
	   step_startTime[11]:= F_GetSystemTime();
	    step_time_seq:=0;
   END_IF
END_IF
END_CASE

///// time update ///////
 
Time_diff[1] := ULINT_TO_UDINT(step_startTime[2]-step_startTime[1])/10000;
Time_diff[2] := ULINT_TO_UDINT(step_startTime[3]-step_startTime[2])/10000; 
Time_diff[3] := ULINT_TO_UDINT(step_startTime[4]-step_startTime[3])/10000;
Time_diff[4] := ULINT_TO_UDINT(step_startTime[5]-step_startTime[4])/10000;
Time_diff[5] := ULINT_TO_UDINT(step_startTime[6]-step_startTime[5])/10000;
Time_diff[6] := ULINT_TO_UDINT(step_startTime[7]-step_startTime[6])/10000;
Time_diff[7] := ULINT_TO_UDINT(step_startTime[8]-step_startTime[7])/10000;
Time_diff[8] := ULINT_TO_UDINT(step_startTime[9]-step_startTime[8])/10000;
Time_diff[9] := ULINT_TO_UDINT(step_startTime[10]-step_startTime[9])/10000;
Time_diff[10] := ULINT_TO_UDINT(step_startTime[11]-step_startTime[10])/10000;

step_time := Time_diff;

END_FUNCTION_BLOCK

// ---- POUs/Programs/OP140/OP140_AutoSequence_2.TcPOU
PROGRAM OP140_AutoSequence_2
VAR 
    OP140_STN_MOVER_2: INT;
	OP140_AutoSeq_2:INT;
	Leak2_FB: OP140_LeakTesting;
	LK2_TS1_Seq_Start: BOOL;
	LK2_TS1_Seq_Completed: BOOL;
	LK2_TS1_tst1_OK: BOOL;
	LK2_TS1_tst1_NOK: BOOL;
	LK2_TS1_tst2_OK: BOOL;
	LK2_TS1_tst2_NOK: BOOL;
	LK2_TS1_tst1_Result: STRING;
	LK2_TS1_tst2_Result: STRING;
	LK2_TS1_CompOK: BOOL;
	LK2_TS1_CompNOK: BOOL;
	LK2_TS2_Seq_Start: BOOL;
	LK2_TS2_Seq_Completed: BOOL;
	LK2_TS2_tst1_OK: BOOL;
	LK2_TS2_tst1_NOK: BOOL;
	LK2_TS2_tst2_OK: BOOL;
	LK2_TS2_tst2_NOK: BOOL;
	LK2_TS2_tst1_Result: STRING;
	LK2_TS2_tst2_Result: STRING;
	LK2_TS2_CompOK: BOOL;
	LK2_TS2_CompNOK: BOOL;
	OP140_Leak2_TS2_result_OK: BOOL;
	OP140_Leak2_TS2_result_NOK: BOOL;
	OP140_Leak2_TS2_Result_Data: STRING;
	OP140_DoneDly_2 : TON;
	OP140_STN_MOVER_2_1: INT;
	OP140_RH_AutoSeq_1: INT;
	CR140_Horz_Cyl_: INT;
	fix_lh_2: INT ;
	fix_rh_2:INT;
	Dry_run : BOOL;
	PRC_DONE	:TON;
END_VAR
VAR
	OP140_Leak2_TS1_result_OK: BOOL;
	OP140_Leak2_TS1_Result_NOK: BOOL;
	OP140_Leak2_TS1_Result_Data: STRING;
	OP1140_LK2_LH_OK: BOOL;
	OP1140_LK2_LH_NOK: BOOL;
	OP1140_LK2_RH_OK: BOOL;
	OP1140_LK2_RH_NOK: BOOL;
END_VAR

IF (NOT OP140_Auto OR  OP140_ErrorActive OR OP140_HomeRunning OR OP140_Machine_Stop ) THEN
	
	OP140_AutoRunning:= FALSE;
	OP140_ComponentOk:=FALSE;
	OP140_ComponentNok:=FALSE;
	OP140_Leak2_Seq_Completed:=FALSE;
	OP140_Leak2_Seq_Start:=FALSE;
	OP140A2_Prev_LH_COMP_OK:=FALSE;
	OP140A2_Prev_RH_COMP_OK:=FALSE;
	OP140_AutoSeq_2:= 10;
	OP140_ATEQ5_ResultOK :=FALSE;
	OP140_ATEQ5_ResultNOK :=FALSE;
	OP140_ATEQ2_ResultOK :=FALSE;
	OP140_ATEQ2_ResultNOK :=FALSE;
	
END_IF

CASE OP140_AutoSeq_2 OF 
	
	10:IF (OP140_Auto) THEN		// Check Automode Selected
		OP140_AutoSeq_2 :=20;
	   END_IF
		
	20:IF ( NOT OP140_ErrorActive) THEN		//Check No error
		OP140_AutoSeq_2:=30;
	   END_IF
	   
	30:IF (NOT OP140_HomeRunning) THEN		//Check No Homerunning
		OP140_AutoSeq_2 :=40;
	   END_IF
		
    40:IF ( OP140_Temp_Home_Ok)THEN	//Check Machine in Home
		OP140_AutoSeq_2:= 50;
		END_IF
		
	50:IF ( NOT OP140_OperationCompleted) AND NOT OP140_TOOL_CHANGE_MODE_SELECTED THEN		// Check Operation Completed Reset
		OP140_AutoSeq_2:=60;
		END_IF
		
	60:IF (NOT OP140_ComponentOk) THEN		// Check Component Ok Reset
		OP140_AutoSeq_2:=70;
		END_IF
		
	70:IF (NOT OP140_ComponentNok) THEN 	// Check Component NOk Reset
		OP140_AutoSeq_2:= 120;
		END_IF
		
    120:IF  ( OP140_HMI_Cycle_Start ) THEN		//Machine Start in Fully Automatic or Press Cycle Start For Semi Automatic
		     OP140_HomeConditionOK:=TRUE;
	 		 IF( OP140_HomeConditionOK AND OP140_AutoSelected) THEN
				OP140_AutoRunning:=TRUE;
				OP140_StepRunning:= FALSE;
				
		     ELSIF ( OP140_HomeConditionOK AND OP140_StepSelected) THEN
					OP140_AutoRunning:=FALSE;
					OP140_StepRunning:= TRUE;
			 END_IF;
		 END_IF
		 
		 IF ((OP140_AutoRunning OR OP140_StepRunning) AND OP140_StartEnable_2)AND  (OP140_DryRun OR OP140_HMI_Cycle_Start)   THEN
              OP140_AutoSeq_2:= 130;
		 END_IF
		 
	130:IF  OP140_STN_ENABLE_2 THEN 
 			OP140_AutoSeq_2:= 140;
		END_IF
		
	140: IF fix_lh_2 <> 130 AND fix_rh_2 <> 130 THEN
		    OP140_AutoSeq_2 := 200;
		 ELSE 
			IF fix_lh_2 =130 AND fix_rh_2 =130 THEN
			   OP140A2_Prev_LH_COMP_OK := TRUE;
	           OP140A2_Prev_RH_COMP_OK := TRUE;
			   OP140_AutoSeq_2 := 150;
			   
			ELSIF fix_lh_2 =130 AND fix_rh_2 =131 THEN
				OP140A2_Prev_LH_COMP_OK := TRUE;
	            OP140A2_Prev_RH_COMP_OK := FALSE;
				OP140_AutoSeq_2 := 150;
				
			ELSIF fix_lh_2 =131 AND fix_rh_2 =130 THEN
				OP140A2_Prev_LH_COMP_OK := FALSE;
	            OP140A2_Prev_RH_COMP_OK :=TRUE ;	
				OP140_AutoSeq_2 := 150;
			END_IF
		END_IF
		
			
	150:IF OP140_StartEnable_2  THEN
		 OP140_Leak2_Seq_Start:=TRUE;	
		 OP140_AutoSeq_2:= 160;
		END_IF
		 
		 
	160:IF OP140_Leak2_Seq_Completed=TRUE  AND In_Range(SR140_Vert_Servo_Ctrl_2.Actual_Position,40,1) THEN
		  OP140A2_LH_Comp_OK:=OP1140_LK2_LH_OK;
		  OP140A2_LH_Comp_NOK:=OP1140_LK2_LH_NOK;
		  OP140A2_RH_Comp_OK:=OP1140_LK2_RH_OK;
		  OP140A2_RH_Comp_NOK:=OP1140_LK2_RH_NOK;
		  OP140_AutoSeq_2:= 170;		
	    END_IF
		OP140_P2_CURR_MVR			:= OP140_STN_MOVER_2;
		
	170: IF OP140_DoneDly_2.q AND OP140_StartEnable THEN
		    
            IF OP140A2_LH_Comp_OK AND OP140A2_RH_Comp_OK THEN
		       MOVER_CMP_STATUS[OP140_P2_CURR_MVR][1]:=142;
		       MOVER_CMP_STATUS[OP140_P2_CURR_MVR][2]:=142;		
			   
		       IF MOVER_CMP_STATUS[OP140_P2_CURR_MVR][1]=142 AND MOVER_CMP_STATUS[OP140_P2_CURR_MVR][2]=142 THEN
				 STATION_DONE[OP140_P2_CURR_MVR][OP140_XTS_POS_NO]			:= TRUE;
				  OP140_AutoSeq_2:= 180;
		       END_IF 	
				
             ELSIF OP140A2_LH_Comp_NOK AND OP140A2_RH_Comp_NOK  THEN
				   MOVER_CMP_STATUS[OP140_P2_CURR_MVR][1]:=143;
		           MOVER_CMP_STATUS[OP140_P2_CURR_MVR][2]:=143;
		
		         IF MOVER_CMP_STATUS[OP140_P2_CURR_MVR][1]=143 AND MOVER_CMP_STATUS[OP140_P2_CURR_MVR][2]=143 THEN
				STATION_DONE[OP140_P2_CURR_MVR][OP140_XTS_POS_NO]			:= TRUE;
				    OP140_AutoSeq_2:= 180;
		         END_IF 
				
             ELSIF OP140A2_LH_Comp_OK AND OP140A2_RH_Comp_NOK  THEN
				   MOVER_CMP_STATUS[OP140_P2_CURR_MVR][1]:=142;
		           MOVER_CMP_STATUS[OP140_P2_CURR_MVR][2]:=143;	
	
		           IF MOVER_CMP_STATUS[OP140_P2_CURR_MVR][1]=142 AND MOVER_CMP_STATUS[OP140_P2_CURR_MVR][2]=143 THEN
				 STATION_DONE[OP140_P2_CURR_MVR][OP140_XTS_POS_NO]			:= TRUE;
				      OP140_AutoSeq_2:= 180;
		           END_IF 	
				
			ELSIF OP140A2_LH_Comp_NOK AND OP140A2_RH_Comp_OK  THEN
				  MOVER_CMP_STATUS[OP140_P2_CURR_MVR][1]:=143;
		          MOVER_CMP_STATUS[OP140_P2_CURR_MVR][2]:=142;		
		         IF MOVER_CMP_STATUS[OP140_P2_CURR_MVR][1]=143 AND MOVER_CMP_STATUS[OP140_P2_CURR_MVR][2]=142 THEN
				STATION_DONE[OP140_P2_CURR_MVR][OP140_XTS_POS_NO]			:= TRUE;
				    OP140_AutoSeq_2:= 180;
		        END_IF 		
		    END_IF		
	     END_IF
	
	180:// Reset All Bits
	
		OP140_Leak2_Seq_Completed:=FALSE;					
        OP140A2_LH_Comp_OK:=FALSE;
        OP140A2_LH_Comp_NOK:=FALSE;
        OP140A2_RH_Comp_OK:=FALSE;
        OP140A2_RH_Comp_NOK:=FALSE;
        OP140_ATEQ5_ResultOK :=FALSE;
		OP140_ATEQ5_ResultNOK :=FALSE;
		OP140_ATEQ2_ResultOK :=FALSE;
		OP140_ATEQ2_ResultNOK :=FALSE;
		OP140_STN_ENABLE_2:=0;
		OP140_AutoSeq_2:= 130;	

	200:MOVER_CMP_STATUS[OP140_P2_CURR_MVR][2]:=143;
		MOVER_CMP_STATUS[OP140_P2_CURR_MVR][1]:=143;
		
		IF MOVER_CMP_STATUS[OP140_P2_CURR_MVR][1]=143 AND MOVER_CMP_STATUS[OP140_P2_CURR_MVR][2]=143 THEN
		STATION_DONE[OP140_STN_MOVER_2][OP140_XTS_POS_NO]			:= TRUE;
		   OP140_AutoSeq_2:= 180;
		END_IF		

END_CASE




Leak2_FB(
	Horz_Cyl_Pos1            := CR140_Horz_Cyl_2.Position1, 
	Horz_Cyl_Pos2            :=CR140_Horz_Cyl_2.Position2 , 
	Vert_Cyl_Pos1            := CR140_Vert_Cyl_2.Position1, 
	Vert_Cyl_Pos2            := CR140_Vert_Cyl_2.Position2, 
	StartEnable              :=OP140_StartEnable_2 , 
	Home_pos_IP              :=OP140_HMI_Vert_Home_Pos, 
	Home_Vel_IP              := OP140_HMI_Vert_Home_Vel,
	SafeHome_Pos_IP          :=OP140_HMI_Vert_SafeHome_Pos,
	SafeHome_Vel_Ip          :=OP140_HMI_Vert_SafeHome_Vel, 
	SafeWork_Pos_IP          :=OP140_HMI_Vert_SafeWork_Pos,
	SafeWork_Vel_IP          :=OP140_HMI_Vert1_SafeWork_Vel,
	Work_Pos_IP              :=OP140_HMI_Vert2_Work_Pos , 
	Work_Vel_IP              :=OP140_HMI_Vert2_Work_Vel , 
	Axis_In_WorkPos          :=SR140_Vert_Servo_Ctrl_2.Axis_In_Pos , 
	Axis_In_Home             :=SR140_Vert_Servo_Ctrl_2.Axis_In_Home , 
	axis_in_position         :=SR140_Vert_Servo_Ctrl_2.Axis_In_Pos,
	servo_actual_pos         :=SR140_Vert_Servo_Ctrl_2.Actual_Position,
	Prev_Stat_LH_OK          :=OP140A2_Prev_LH_COMP_OK , 
	Prev_Stat_RH_OK          :=OP140A2_Prev_RH_COMP_OK , 
	TS1_Test1_ProgNO         :=OP140_ATEQ_Test_Prog1_No , 
	TS1_Test2_ProgNO         :=OP140_ATEQ_Test_Prog2_No , 
	TS1_TestOk               :=OP140_ATEQ2_ResultOK , 
	TS1_TestNOK              :=OP140_ATEQ2_ResultNOK , 
	TS1_StartEnable          := OP140_StartEnable_2, 
	TS1_ResultIN             := OP140_ATEQ2_Result , 
	TS2_Test1_ProgNO         :=OP140_ATEQ_Test_Prog1_No , 
	TS2_Test2_ProgNO         :=OP140_ATEQ_Test_Prog2_No , 
	TS2_TestOk               :=OP140_ATEQ5_ResultOK , 
	TS2_TestNOK              :=OP140_ATEQ5_ResultNOK , 
	TS2_StartEnable          :=OP140_StartEnable_2 , 
	TS2_ResultIN             :=OP140_ATEQ5_Result , 
	Horz_Cyl_Auto1            =>CR140_Horz_Cyl_2.AutoCmd1 , 
	Horz_Cyl_Auto2            =>CR140_Horz_Cyl_2.AutoCmd2 , 
	Vert_Cyl_Auto1            =>CR140_Vert_Cyl_2.AutoCmd1 , 
	Vert_Cyl_Auto2            =>CR140_Vert_Cyl_2.AutoCmd2 , 
	Servo_Pos_Error           => , 
	Servo_HomePos_Error       => , 
	TS1_StartOP               => OP140_ATEQ2_Auto_Start , 
	TS1_Test_ProgNO           => OP140_ATEQ2_Auto_Prog_No_out , 
	TS2_StartOP               =>OP140_ATEQ5_Auto_Start , 
	TS2_Test_ProgNO           => OP140_ATEQ5_Auto_Prog_No_out , 
	Seq_Start                 := OP140_Leak2_Seq_Start, 
	Seq_Completed             :=OP140_Leak2_Seq_Completed , 
	TS1_SeqStart              :=LK2_TS1_Seq_Start , 
	TS1_SeqCompleted          := LK2_TS1_Seq_Completed, 
	TS1_ATEQCompleted         :=  OP140_ATEQ2_ResultCompleted, 
	TS1_Test1OK               :=LK2_TS2_tst1_OK , 
	TS1_Test1NOK              := LK2_TS1_tst1_NOK, 
	TS1_Test2Ok               :=LK2_TS1_tst2_OK , 
	TS1_Test2NOK              :=LK2_TS1_tst2_NOK , 
	TS1_Test1Result           := LK2_TS1_tst1_Result, 
	TS1_Test2Result           :=LK2_TS1_tst2_Result , 
	TS1_CompOK                :=LK2_TS1_CompOK , 
	TS1_CompNOK               := LK2_TS1_CompNOK, 
	TS1_ResultOK              :=OP140_Leak2_TS1_result_OK , 
	TS1_ResultNOK             := OP140_Leak2_TS1_Result_NOK, 
	TS1_Result_Data           :=OP140_Leak2_TS1_Result_Data , 
	LH_CompOK                 :=OP1140_LK2_LH_OK , 
	LH_CompNOK                :=OP1140_LK2_LH_NOK , 
	RH_CompOK                 :=OP1140_LK2_RH_OK , 
	RH_CompNOK                :=OP1140_LK2_RH_NOK , 
	TS2_SeqStart              :=LK2_TS2_Seq_Start , 
	TS2_SeqCompleted          := LK2_TS2_Seq_Completed , 
	TS2_ATEQCompleted         :=OP140_ATEQ5_ResultCompleted , 
	TS2_Test1OK               :=LK2_TS2_tst1_OK , 
	TS2_Test1NOK              :=LK2_TS2_tst1_NOK  , 
	TS2_Test2Ok               :=LK2_TS2_tst2_OK , 
	TS2_Test2NOK              :=LK2_TS2_tst2_NOK , 
	TS2_Test1Result           := LK2_TS2_tst1_Result , 
	TS2_Test2Result           :=LK2_TS2_tst2_Result , 
	TS2_CompOK                :=LK2_TS2_CompOK , 
	TS2_CompNOK               :=LK2_TS2_CompNOK , 
	TS2_ResultOK              := OP140_Leak2_TS2_result_OK, 
	TS2_ResultNOK             :=OP140_Leak2_TS2_result_NOK , 
	TS2_Result_Data           :=OP140_Leak2_TS2_Result_Data ,
    Servo_Pos_OP              :=SR140_Vert_Servo_Ctrl_2.Position,
    Servo_Vel_OP              :=SR140_Vert_Servo_Ctrl_2.Velocity,
    ABS_Move_Start            :=SR140_Vert_Servo_Ctrl_2.ABSmove_Start);

OP140_DoneDly_2(IN:=OP140_Leak2_Seq_Completed , PT:=T#500MS , Q=> , ET=> );
dry_run:=All_Station_Dry_Run;	
IF Dry_Run THEN
	fix_lh_2:=130;	
    fix_rh_2:=130;
ELSE
	fix_lh_2:=MOVER_CMP_STATUS[OP140_STN_MOVER_2][1];	
    fix_rh_2:=MOVER_CMP_STATUS[OP140_STN_MOVER_2][2];	
END_IF
	

//############################		OP140 STATION ENABLE CONDITION		##########################

OP140_STN_MOVER_2					:= MOVER_POSITION[OP140_P2_XTS_POS_NO];

IF AUTO_WITH_XTS THEN
IF OP140_STN_MOVER_2>0 THEN
IF NOT(END_OF_CYCLE AND MOVER_CMP_STATUS[OP140_STN_MOVER_2][1]=5 AND MOVER_CMP_STATUS[OP140_STN_MOVER_2][2]=5)THEN
OP140_STN_ENABLE_2					:= MOVER_POS_RECHED[OP140_STN_MOVER_2] AND ((MOVER_CMP_STATUS[OP140_STN_MOVER_2][1]=130)OR 
									(MOVER_CMP_STATUS[OP140_STN_MOVER_2][2]=130))AND STATION_ENABLE_CONTROL;
ELSE
	STATION_DONE[OP140_STN_MOVER_2][OP140_XTS_POS_NO]			:= TRUE;
END_IF
ELSE
OP140_STN_ENABLE_2					:= FALSE;
END_IF	
END_IF

END_PROGRAM

// ---- POUs/Programs/OP140/OP140_AutoSequence_3.TcPOU
PROGRAM OP140_AutoSequence_3
VAR
	OP140_AutoSeq_3:INT;

	OP140_STN_MOVER_3: INT;
	
	Leak3_FB: OP140_LeakTesting;
	LK3_TS1_Seq_Start: BOOL;
	LK3_TS1_Seq_Completed: BOOL;
	LK3_TS1_tst1_OK: BOOL;
	LK3_TS1_tst1_NOK: BOOL;
	LK3_TS1_tst2_OK: BOOL;
	LK3_TS1_tst2_NOK: BOOL;
	LK3_TS1_tst1_Result: STRING;
	LK3_TS1_tst2_Result: STRING;
	LK3_TS1_CompOK: BOOL;
	LK3_TS1_CompNOK: BOOL;	
	LK3_TS2_Seq_Start: BOOL;
	LK3_TS2_Seq_Completed: BOOL;
	LK3_TS2_tst1_OK: BOOL;
	LK3_TS2_tst1_NOK: BOOL;
	LK3_TS2_tst2_OK: BOOL;
	LK3_TS2_tst2_NOK: BOOL;
	LK3_TS2_tst1_Result: STRING;
	LK3_TS2_tst2_Result: STRING;
	LK3_TS2_CompOK: BOOL;
	LK3_TS2_CompNOK: BOOL;
	OP140_Leak3_TS2_result_OK: BOOL;
	OP140_Leak3_TS2_result_NOK: BOOL;
	OP140_Leak3_TS2_Result_Data: STRING;
	OP140_Stn_EnableTRIG: R_TRIG;
	OP140_DoneDly_3: TON;
	fix_rh_3: INT;
	fix_lh_3: INT;
	Dry_Run: BOOL;
	timeee: Ton;
END_VAR
VAR 
	OP140_Leak3_TS1_result_OK: BOOL;
	OP140_Leak3_TS1_Result_NOK: BOOL;
	OP140_Leak3_TS1_Result_Data: STRING;
	OP1140_LK3_LH_OK: BOOL;
	OP1140_LK3_LH_NOK: BOOL;
	OP1140_LK3_RH_OK: BOOL;
	OP1140_LK3_RH_NOK: BOOL;
END_VAR

IF (NOT OP140_Auto OR  OP140_ErrorActive OR OP140_HomeRunning OR OP140_Machine_Stop ) THEN
	
	OP140_AutoRunning:= FALSE;
	OP140_ComponentOk:=FALSE;
	OP140_ComponentNok:=FALSE;
	OP140_AutoSeq_3:= 10;
	OP140_Leak3_Seq_Completed:=FALSE;
	OP140_Leak3_Seq_Start:=FALSE;
	OP140A3_Prev_LH_COMP_OK:=FALSE;
	OP140A3_Prev_RH_COMP_OK:=FALSE;
	OP140_ATEQ1_ResultOK :=FALSE;
	OP140_ATEQ1_ResultNOK :=FALSE;
	OP140_ATEQ4_ResultOK :=FALSE;
	OP140_ATEQ4_ResultNOK :=FALSE;
	
END_IF

CASE OP140_AutoSeq_3 OF 
	
	10:IF (OP140_Auto) THEN		// Check Automode Selected
		  OP140_AutoSeq_3 :=20;
	   END_IF
	   
	20:IF ( NOT OP140_ErrorActive) THEN		//Check No error
		  OP140_AutoSeq_3:=30;
	   END_IF
	   
	30:IF (NOT OP140_HomeRunning) THEN		//Check No Homerunning
		  OP140_AutoSeq_3 :=40;
	   END_IF
	   
    40:IF ( OP140_Temp_Home_Ok)THEN	//Check Machine in Home
		OP140_AutoSeq_3:= 50;
	   END_IF
		
	50:IF ( NOT OP140_OperationCompleted) AND NOT OP140_TOOL_CHANGE_MODE_SELECTED THEN		// Check Operation Completed Reset
		OP140_AutoSeq_3:=60;
		END_IF
		
	60:IF (NOT OP140_ComponentOk) THEN		// Check Component Ok Reset
		OP140_AutoSeq_3:=70;
	   END_IF
		
	70:IF (NOT OP140_ComponentNok) THEN 	// Check Component NOk Reset
		OP140_AutoSeq_3:= 120;
	   END_IF
		
    120:IF  ( OP140_HMI_Cycle_Start ) THEN		//Machine Start in Fully Automatic or Press Cycle Start For Semi Automatic
		     OP140_HomeConditionOK:=TRUE;
			 IF( OP140_HomeConditionOK AND OP140_AutoSelected) THEN
			    OP140_AutoRunning:=TRUE;
				OP140_StepRunning:= FALSE;
			 ELSIF ( OP140_HomeConditionOK AND OP140_StepSelected) THEN
					OP140_AutoRunning:=FALSE;
					OP140_StepRunning:= TRUE;
				END_IF;
		 END_IF
		 
		 IF ((OP140_AutoRunning OR OP140_StepRunning) AND OP140_StartEnable_1)AND  (OP140_DryRun OR OP140_HMI_Cycle_Start)   THEN
              OP140_AutoSeq_3:= 130;
		END_IF
		
	130:IF  OP140_STN_ENABLE_3 THEN 
 			OP140_AutoSeq_3:= 140;
			
		ELSIF NOT OP140_STN_ENABLE_3 AND  MOVER_POS_RECHED[OP140_STN_MOVER_3] AND fix_lh_3 <> 130 AND fix_rh_3 <> 130 THEN
				OP140_AutoSeq_3 := 200;
		END_IF
		
	140:    IF fix_lh_3 =130 AND fix_rh_3 =130 THEN
			   OP140A3_Prev_LH_COMP_OK := TRUE;
	           OP140A3_Prev_RH_COMP_OK := TRUE;
			   OP140_AutoSeq_3 := 150;
			   
			ELSIF fix_lh_3 =130 AND fix_rh_3 =131 THEN
				OP140A3_Prev_LH_COMP_OK := TRUE;
	            OP140A3_Prev_RH_COMP_OK := FALSE;
				OP140_AutoSeq_3 := 150;
				
			ELSIF fix_lh_3 =131 AND fix_rh_3 =130 THEN
				OP140A3_Prev_LH_COMP_OK := FALSE;
	            OP140A3_Prev_RH_COMP_OK :=TRUE ;
	            OP140_AutoSeq_3 := 150;
			END_IF
			

	150:IF OP140_StartEnable_3  THEN
		 OP140_Leak3_Seq_Start:=TRUE;	
		 OP140_AutoSeq_3:= 160;
		END_IF
		 
		 
	160:IF OP140_Leak3_Seq_Completed=TRUE AND In_Range(SR140_Vert_Servo_Ctrl_3.Actual_Position,40,1)  THEN
		  OP140A3_LH_Comp_OK:=OP1140_LK3_LH_OK;
		  OP140A3_LH_Comp_NOK:=OP1140_LK3_LH_NOK;
		  OP140A3_RH_Comp_OK:=OP1140_LK3_RH_OK;
		  OP140A3_RH_Comp_NOK:=OP1140_LK3_RH_NOK;
		  OP140_AutoSeq_3:= 170;		
	    END_IF
		OP140_P3_CURR_MVR 					:= OP140_STN_MOVER_3;
	170: IF OP140_DoneDly_3.q AND OP140_StartEnable THEN
		    IF OP140A3_LH_Comp_OK AND OP140A3_RH_Comp_OK THEN
		       MOVER_CMP_STATUS[OP140_P3_CURR_MVR][1]:=144;
		       MOVER_CMP_STATUS[OP140_P3_CURR_MVR][2]:=144;
		
		       IF MOVER_CMP_STATUS[OP140_P3_CURR_MVR][1]=144 AND MOVER_CMP_STATUS[OP140_P3_CURR_MVR][2]=144 THEN
				   STATION_DONE[OP140_P3_CURR_MVR][OP140_XTS_POS_NO]			:= TRUE;
				  OP140_AutoSeq_3:= 180;
		        END_IF 	
				
             ELSIF OP140A3_LH_Comp_NOK AND OP140A3_RH_Comp_NOK  THEN
				 MOVER_CMP_STATUS[OP140_P3_CURR_MVR][1]:=145;
		         MOVER_CMP_STATUS[OP140_P3_CURR_MVR][2]:=145;
		
		         IF MOVER_CMP_STATUS[OP140_P3_CURR_MVR][1]=145 AND MOVER_CMP_STATUS[OP140_P3_CURR_MVR][2]=145 THEN
				    STATION_DONE[OP140_P3_CURR_MVR][OP140_XTS_POS_NO]			:= TRUE;
				    OP140_AutoSeq_3:= 180;
		        END_IF 
				
             ELSIF OP140A3_LH_Comp_OK AND OP140A3_RH_Comp_NOK  THEN
				   MOVER_CMP_STATUS[OP140_P3_CURR_MVR][1]:=144;
		           MOVER_CMP_STATUS[OP140_P3_CURR_MVR][2]:=145;	
	
		         IF MOVER_CMP_STATUS[OP140_P3_CURR_MVR][1]=144 AND MOVER_CMP_STATUS[OP140_P3_CURR_MVR][2]=145 THEN
				  STATION_DONE[OP140_P3_CURR_MVR][OP140_XTS_POS_NO]			:= TRUE;
				    OP140_AutoSeq_3:= 180;
		        END_IF 	
				
			ELSIF OP140A3_LH_Comp_NOK AND OP140A3_RH_Comp_OK  THEN
				  MOVER_CMP_STATUS[OP140_P3_CURR_MVR][1]:=145;
		          MOVER_CMP_STATUS[OP140_P3_CURR_MVR][2]:=144;	
	
		         IF MOVER_CMP_STATUS[OP140_P3_CURR_MVR][1]=145 AND MOVER_CMP_STATUS[OP140_P3_CURR_MVR][2]=144 THEN
			STATION_DONE[OP140_P3_CURR_MVR][OP140_XTS_POS_NO]			:= TRUE;
				    OP140_AutoSeq_3:= 180;
		        END_IF 		
		    END_IF		
	     END_IF
	
	180:// Reset All Bits
		
 		OP140_Leak3_Seq_Completed:=FALSE;					
        OP140A3_LH_Comp_OK:=FALSE;
        OP140A3_LH_Comp_NOK:=FALSE;
        OP140A3_RH_Comp_OK:=FALSE;
        OP140A3_RH_Comp_NOK:=FALSE; 
		OP140_ATEQ1_ResultOK :=FALSE;
		OP140_ATEQ1_ResultNOK :=FALSE;
		OP140_ATEQ4_ResultOK :=FALSE;
		OP140_ATEQ4_ResultNOK :=FALSE;
		OP140_STN_ENABLE_3:=0;
		OP140_AutoSeq_3:= 130;	

	200:MOVER_CMP_STATUS[OP140_P3_CURR_MVR][2]:=140;
		MOVER_CMP_STATUS[OP140_P3_CURR_MVR][1]:=140;
		
		IF MOVER_CMP_STATUS[OP140_P3_CURR_MVR][1]=140 AND MOVER_CMP_STATUS[OP140_P3_CURR_MVR][2]=140 THEN
		 STATION_DONE[OP140_STN_MOVER_3][OP140_XTS_POS_NO]			:= TRUE;
		   OP140_AutoSeq_3:= 180;
		END_IF		

END_CASE

//Leak3FB

Leak3_FB(
	
	Horz_Cyl_Pos1                 := CR140_Horz_Cyl_3.Position1, 
	Horz_Cyl_Pos2                 :=CR140_Horz_Cyl_3.Position2 , 
	Vert_Cyl_Pos1                 := CR140_Vert_Cyl_3.Position1, 
	Vert_Cyl_Pos2                 := CR140_Vert_Cyl_3.Position2, 
	StartEnable                   :=OP140_StartEnable_3 , 
	Home_pos_IP                   :=OP140_HMI_Vert_Home_Pos , 
	Home_Vel_IP                   := OP140_HMI_Vert_Home_Vel, 
	SafeHome_Pos_IP               :=OP140_HMI_Vert_SafeHome_Pos,
	SafeHome_Vel_Ip               :=OP140_HMI_Vert_SafeHome_Vel,
	SafeWork_Pos_IP               :=OP140_HMI_Vert_SafeWork_Pos,
	SafeWork_Vel_IP               :=OP140_HMI_Vert1_SafeWork_Vel,
	Work_Pos_IP                   :=OP140_HMI_Vert3_Work_Pos , 
	Work_Vel_IP                   :=OP140_HMI_Vert3_Work_Vel , 
	Axis_In_WorkPos               :=SR140_Vert_Servo_Ctrl_3.Axis_In_Pos , 
	Axis_In_Home                  :=SR140_Vert_Servo_Ctrl_3.Axis_In_Home , 
	axis_in_position              :=SR140_Vert_Servo_Ctrl_3.Axis_In_Pos,
	servo_actual_pos              :=SR140_Vert_Servo_Ctrl_3.Actual_Position,	
	Prev_Stat_LH_OK               :=OP140A3_Prev_LH_COMP_OK , 
	Prev_Stat_RH_OK               :=OP140A3_Prev_RH_COMP_OK , 
	TS1_Test1_ProgNO              :=OP140_ATEQ_Test_Prog1_No , 
	TS1_Test2_ProgNO              :=OP140_ATEQ_Test_Prog2_No , 
	TS1_TestOk                    :=OP140_ATEQ1_ResultOK , 
	TS1_TestNOK                   :=OP140_ATEQ1_ResultNOK , 
	TS1_StartEnable               := OP140_StartEnable_3, 
	TS1_ResultIN                  := OP140_ATEQ1_Result , 
	TS2_Test1_ProgNO              :=OP140_ATEQ_Test_Prog1_No , 
	TS2_Test2_ProgNO              :=OP140_ATEQ_Test_Prog2_No , 
	TS2_TestOk                    :=OP140_ATEQ4_ResultOK , 
	TS2_TestNOK                   :=OP140_ATEQ4_ResultNOK , 
	TS2_StartEnable               :=OP140_StartEnable_3 , 
	TS2_ResultIN                  :=OP140_ATEQ4_Result , 
	Horz_Cyl_Auto1                =>CR140_Horz_Cyl_3.AutoCmd1 , 
	Horz_Cyl_Auto2                =>CR140_Horz_Cyl_3.AutoCmd2 , 
	Vert_Cyl_Auto1                =>CR140_Vert_Cyl_3.AutoCmd1 , 
	Vert_Cyl_Auto2                =>CR140_Vert_Cyl_3.AutoCmd2 , 
	Servo_Pos_Error               => , 
	Servo_HomePos_Error           => , 
	TS1_StartOP                   => OP140_ATEQ1_Auto_Start , 
	TS1_Test_ProgNO               => OP140_ATEQ1_Auto_Prog_No_out , 
	TS2_StartOP                   => OP140_ATEQ4_Auto_Start , 
	TS2_Test_ProgNO               => OP140_ATEQ4_Auto_Prog_No_out , 
	Seq_Start                     := OP140_Leak3_Seq_Start, 
	Seq_Completed                 := OP140_Leak3_Seq_Completed , 
	TS1_SeqStart                  := LK3_TS1_Seq_Start , 
	TS1_SeqCompleted              := LK3_TS1_Seq_Completed, 
	TS1_ATEQCompleted             := OP140_ATEQ1_ResultCompleted, 
	TS1_Test1OK                   := LK3_TS1_tst1_OK , 
	TS1_Test1NOK                  := LK3_TS1_tst1_NOK, 
	TS1_Test2Ok                   := LK3_TS1_tst2_OK , 
	TS1_Test2NOK                  := LK3_TS1_tst2_NOK , 
	TS1_Test1Result               := LK3_TS1_tst1_Result, 
	TS1_Test2Result               := LK3_TS1_tst2_Result , 
	TS1_CompOK                    := LK3_TS1_CompOK , 
	TS1_CompNOK                   := LK3_TS1_CompNOK, 
	TS1_ResultOK                  := OP140_Leak3_TS1_result_OK , 
	TS1_ResultNOK                 := OP140_Leak3_TS1_Result_NOK, 
	TS1_Result_Data               := OP140_Leak3_TS1_Result_Data , 
	LH_CompOK                     := OP1140_LK3_LH_OK , 
	LH_CompNOK                    := OP1140_LK3_LH_NOK , 
	RH_CompOK                     := OP1140_LK3_RH_OK , 
	RH_CompNOK                    := OP1140_LK3_RH_NOK , 
	TS2_SeqStart                  := LK3_TS2_Seq_Start , 
	TS2_SeqCompleted              := LK3_TS2_Seq_Completed , 
	TS2_ATEQCompleted             :=OP140_ATEQ4_ResultCompleted , 
	TS2_Test1OK                   :=LK3_TS2_tst1_OK , 
	TS2_Test1NOK                  :=LK3_TS2_tst1_NOK  , 
	TS2_Test2Ok                   :=LK3_TS2_tst2_OK , 
	TS2_Test2NOK                  :=LK3_TS2_tst2_NOK , 
	TS2_Test1Result               := LK3_TS2_tst1_Result , 
	TS2_Test2Result               :=LK3_TS2_tst2_Result , 
	TS2_CompOK                    :=LK3_TS2_CompOK , 
	TS2_CompNOK                   :=LK3_TS2_CompNOK , 
	TS2_ResultOK                  := OP140_Leak3_TS2_result_OK, 
	TS2_ResultNOK                 :=OP140_Leak3_TS2_result_NOK , 
	TS2_Result_Data               :=OP140_Leak3_TS2_Result_Data ,
    Servo_Pos_OP                  :=SR140_Vert_Servo_Ctrl_3.Position,
    Servo_Vel_OP                  :=SR140_Vert_Servo_Ctrl_3.Velocity,
    ABS_Move_Start                :=SR140_Vert_Servo_Ctrl_3.ABSmove_Start);

	
OP140_DoneDly_3(IN:=OP140_Leak3_Seq_Completed , PT:=T#500MS , Q=> , ET=> );
	
dry_run:=All_Station_Dry_Run;	
IF Dry_Run THEN
	fix_lh_3:=130;	
    fix_rh_3:=130;
ELSE
	fix_lh_3:=MOVER_CMP_STATUS[OP140_STN_MOVER_3][1];	
    fix_rh_3:=MOVER_CMP_STATUS[OP140_STN_MOVER_3][2];	
END_IF


//############################		OP140 STATION ENABLE CONDITION		##########################

	OP140_STN_MOVER_3					:= MOVER_POSITION[OP140_P3_XTS_POS_NO];
	
	IF AUTO_WITH_XTS THEN
	IF OP140_STN_MOVER_3>0 THEN	
	IF NOT(END_OF_CYCLE AND MOVER_CMP_STATUS[OP140_STN_MOVER_3][1]=5 AND MOVER_CMP_STATUS[OP140_STN_MOVER_3][2]=5)THEN
	OP140_STN_ENABLE_3					:= MOVER_POS_RECHED[OP140_STN_MOVER_3] AND ((MOVER_CMP_STATUS[OP140_STN_MOVER_3][1]=130)OR 
										(MOVER_CMP_STATUS[OP140_STN_MOVER_3][2]=130))AND STATION_ENABLE_CONTROL;	
	ELSE
	STATION_DONE[OP140_STN_MOVER_3][OP140_XTS_POS_NO]			:= TRUE;		
	END_IF
	ELSE
	OP140_STN_ENABLE_3					:= FALSE;
	END_IF
	END_IF

END_PROGRAM

// ---- POUs/Programs/OP140/OP140_Error.TcPOU
PROGRAM OP140_Error
VAR
	Step_No: INT;
	AutoStepErr_1: TON;
	OP140_StepErr1: TON;
	OP140_StepErr2: TON;
	bdone: BOOL;
	i: INT;
	j: INT;
END_VAR

IF NOT bdone THEN
	bdone:=TRUE;
FOR i:=1300 TO 1400 BY 1 DO 
	
IF berror[i] THEN
	OP140_ErrorActive:=TRUE;
END_IF
END_FOR
bdone:=FALSE;
END_IF

IF OP130_HMI_Reset OR Servo_Reset THEN
	FOR j:=1300 TO 1400 BY 1 DO 
		
	
	berror[j]:=FALSE;
	OP140_ErrorActive:=FALSE;
	
	END_FOR
	temp:=false;
END_IF

END_PROGRAM

// ---- POUs/Programs/OP140/OP140_Manual.TcPOU
PROGRAM OP140_Manual
VAR
	OP140_Enable:BOOL;
	temp : BOOL;
	temp1: BOOL;
	temp3: BOOL;
END_VAR

//Bottom Cylinder 1
OP140_GVL.CR140_Horz_Cyl_1_Status:=0;
// Safe Home
IF CR140_Vert_Cyl_1.position1 THEN 
	CR140_Horz_Cyl_1.SafeHome:= TRUE;
	ELSE
		CR140_Horz_Cyl_1.SafeHome:= FALSE;
	END_IF
	//Safe Work
IF CR140_Vert_Cyl_1.position1 THEN 
CR140_Horz_Cyl_1.SafeWork:=TRUE;
ELSE
	CR140_Horz_Cyl_1.SafeWork:=FALSE;
	END_IF
//Manual PB 1
IF(OP140_HMI_Horz_Cyl1_Home_PB) THEN
	CR140_Horz_Cyl_1.ManualPB1:=TRUE;
	ELSE
		CR140_Horz_Cyl_1.ManualPB1:=FALSE;
	END_IF
//Manual PB2 
IF(OP140_HMI_Horz_Cyl1_Work_PB) THEN
	CR140_Horz_Cyl_1.ManualPB2:=TRUE;
	ELSE
		CR140_Horz_Cyl_1.ManualPB2:=FALSE;
	END_IF	

	

CR140_Horz_Cyl_1(
	Auto:=OP140_AutoSelected , 
	Manual:=OP140_ManualSelected , 
	ErrorActive:=OP140_ErrorActive , 
	ResetPB:=OP140_HMI_Reset , 
	Sensor1:=I140_HORZ_SUP1_CYL_REVI1301_0  , 
	Sensor2:=I140_HORZ_SUP1_CYL_FWDI1301_1  , 
	ManualPB1:= , 
	ManualPB2:= , 
	AutoCmd1:= , 
	AutoCmd2:= , 
	OperationEnable:=OperationEnable , 
	SafeHome:= , 
	SafeWork:= , 
	HomingCmd1:= , 
	Pulse_1Sec:=Pulse_Block.Q1Hz , 
	BlinkingBit:= , 
	TimeOut1:=10 , 
	TimeOut2:=10 , 
	TimeOut3:=10 , 
	Solenoid1=>O140_HORZ_SUP1_CYL_REV_Q1341_0 , 
	Solenoid2=>O140_HORZ_SUP1_CYL_FWD_Q1341_1 , 
	AlarmSensor1=>berror[1301] , 
	AlarmSensor2=>berror[1302] , 
	AlarmSolenoid1=>berror[1303] , 
	AlarmSolenoid2=> berror[1304], 
	AllSignal=>berror[1305] , 
	AlarmPresent=> , 
	Position1=> , 
	Position2=> , 
	HomeSensorBlink=> , 
	WorkSensorBlink=> , 
	Status:=OP140_GVL.CR140_Horz_Cyl_1_Status );
	
	
	//Bottom Cylinder 2
OP140_GVL.CR140_Horz_Cyl_2_Status:=0;
// Safe Home
IF CR140_Vert_Cyl_2.position1 THEN 
	CR140_Horz_Cyl_2.SafeHome:= TRUE;
	ELSE
		CR140_Horz_Cyl_2.SafeHome:= FALSE;
	END_IF
	//Safe Work
IF CR140_Vert_Cyl_2.position1 THEN 
CR140_Horz_Cyl_2.SafeWork:=TRUE;
ELSE
	CR140_Horz_Cyl_2.SafeWork:=FALSE;
	END_IF
//Manual PB 1
IF(OP140_HMI_Horz_Cyl2_Home_PB) THEN
	CR140_Horz_Cyl_2.ManualPB1:=TRUE;
	ELSE
		CR140_Horz_Cyl_2.ManualPB1:=FALSE;
	END_IF
//Manual PB2 
IF(OP140_HMI_Horz_Cyl2_Work_PB) THEN
	CR140_Horz_Cyl_2.ManualPB2:=TRUE;
	ELSE
		CR140_Horz_Cyl_2.ManualPB2:=FALSE;
	END_IF	

	

CR140_Horz_Cyl_2(
	Auto:= OP140_AutoSelected, 
	Manual:=OP140_ManualSelected , 
	ErrorActive:=OP140_ErrorActive , 
	ResetPB:=OP140_HMI_Reset  , 
	Sensor1:=I140_HORZ_SUP2_CYL_REVI1310_0  , 
	Sensor2:=I140_HORZ_SUP2_CYL_FWDI1310_1  , 
	ManualPB1:= , 
	ManualPB2:= , 
	AutoCmd1:= , 
	AutoCmd2:= , 
	OperationEnable:= OperationEnable, 
	SafeHome:= , 
	SafeWork:= , 
	HomingCmd1:= , 
	Pulse_1Sec:=Pulse_Block.Q1Hz , 
	BlinkingBit:= , 
	TimeOut1:=10 , 
	TimeOut2:=10 , 
	TimeOut3:=10 , 
	Solenoid1=>O140_HORZ_SUP2_CYL_REV_Q1342_0 , 
	Solenoid2=>O140_HORZ_SUP2_CYL_FWD_Q1342_1  , 
	AlarmSensor1=>berror[1316] , 
	AlarmSensor2=>berror[1317] , 
	AlarmSolenoid1=>berror[1318] , 
	AlarmSolenoid2=>berror[1319] , 
	AllSignal=>berror[1320] , 
	AlarmPresent=> , 
	Position1=> , 
	Position2=> , 
	HomeSensorBlink=> , 
	WorkSensorBlink=> , 
	Status:=OP140_GVL.CR140_Horz_Cyl_2_Status);
	
	
	//Bottom Cylinder 3
OP140_GVL.CR140_Horz_Cyl_3_Status:=0;
// Safe Home
IF CR140_Vert_Cyl_3.position1 THEN 
	CR140_Horz_Cyl_3.SafeHome:= TRUE;
	ELSE
		CR140_Horz_Cyl_3.SafeHome:= FALSE;
	END_IF
	//Safe Work
IF CR140_Vert_Cyl_3.position1 THEN 
CR140_Horz_Cyl_3.SafeWork:=TRUE;
ELSE
	CR140_Horz_Cyl_3.SafeWork:=FALSE;
	END_IF
//Manual PB 1
IF(OP140_HMI_Horz_Cyl3_Home_PB) THEN
	CR140_Horz_Cyl_3.ManualPB1:=TRUE;
	ELSE
		CR140_Horz_Cyl_3.ManualPB1:=FALSE;
	END_IF
//Manual PB2 
IF(OP140_HMI_Horz_Cyl3_Work_PB) THEN
	CR140_Horz_Cyl_3.ManualPB2:=TRUE;
	ELSE
		CR140_Horz_Cyl_3.ManualPB2:=FALSE;
	END_IF	

	

